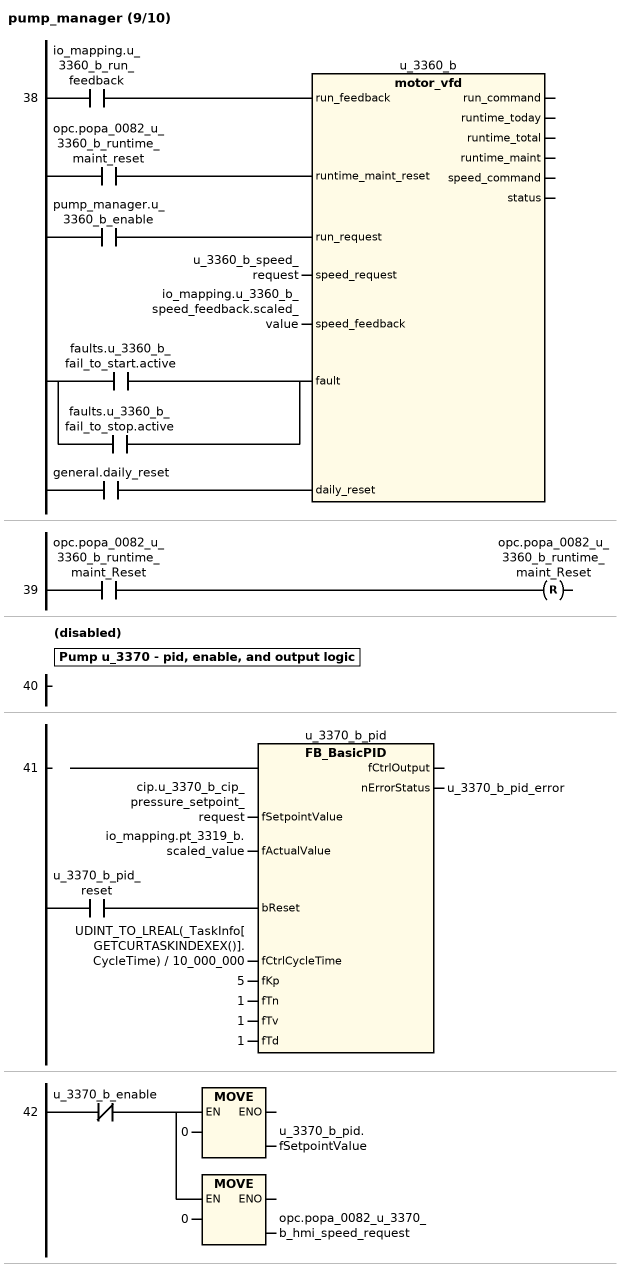
// NETWORK 38
u_3360_b(
    run_feedback := io_mapping.u_3360_b_run_feedback,
    runtime_maint_reset := opc.popa_0082_u_3360_b_runtime_maint_reset,
    run_request := pump_manager.u_3360_b_enable,
    speed_request := u_3360_b_speed_request,
    speed_feedback := io_mapping.u_3360_b_speed_feedback.scaled_value,
    fault := faults.u_3360_b_fail_to_start.active OR faults.u_3360_b_fail_to_stop.active,
    daily_reset := general.daily_reset); // motor_vfd

// NETWORK 39
opc.popa_0082_u_3360_b_runtime_maint_Reset R= opc.popa_0082_u_3360_b_runtime_maint_Reset;

// NETWORK 40 (disabled)
// label: Pump u_3370 - pid, enable, and output logic

// NETWORK 41
u_3370_b_pid(
    fSetpointValue := cip.u_3370_b_cip_pressure_setpoint_request,
    fActualValue := io_mapping.pt_3319_b.scaled_value,
    bReset := u_3370_b_pid_reset,
    fCtrlCycleTime := UDINT_TO_LREAL(_TaskInfo[GETCURTASKINDEXEX()].CycleTime) / 10_000_000,
    fKp := 5,
    fTn := 1,
    fTv := 1,
    fTd := 1,
    nErrorStatus => u_3370_b_pid_error); // FB_BasicPID

// NETWORK 42
_w24 := NOT u_3370_b_enable;
IF _w24 THEN u_3370_b_pid.fSetpointValue := 0; END_IF
IF _w24 THEN opc.popa_0082_u_3370_b_hmi_speed_request := 0; END_IF

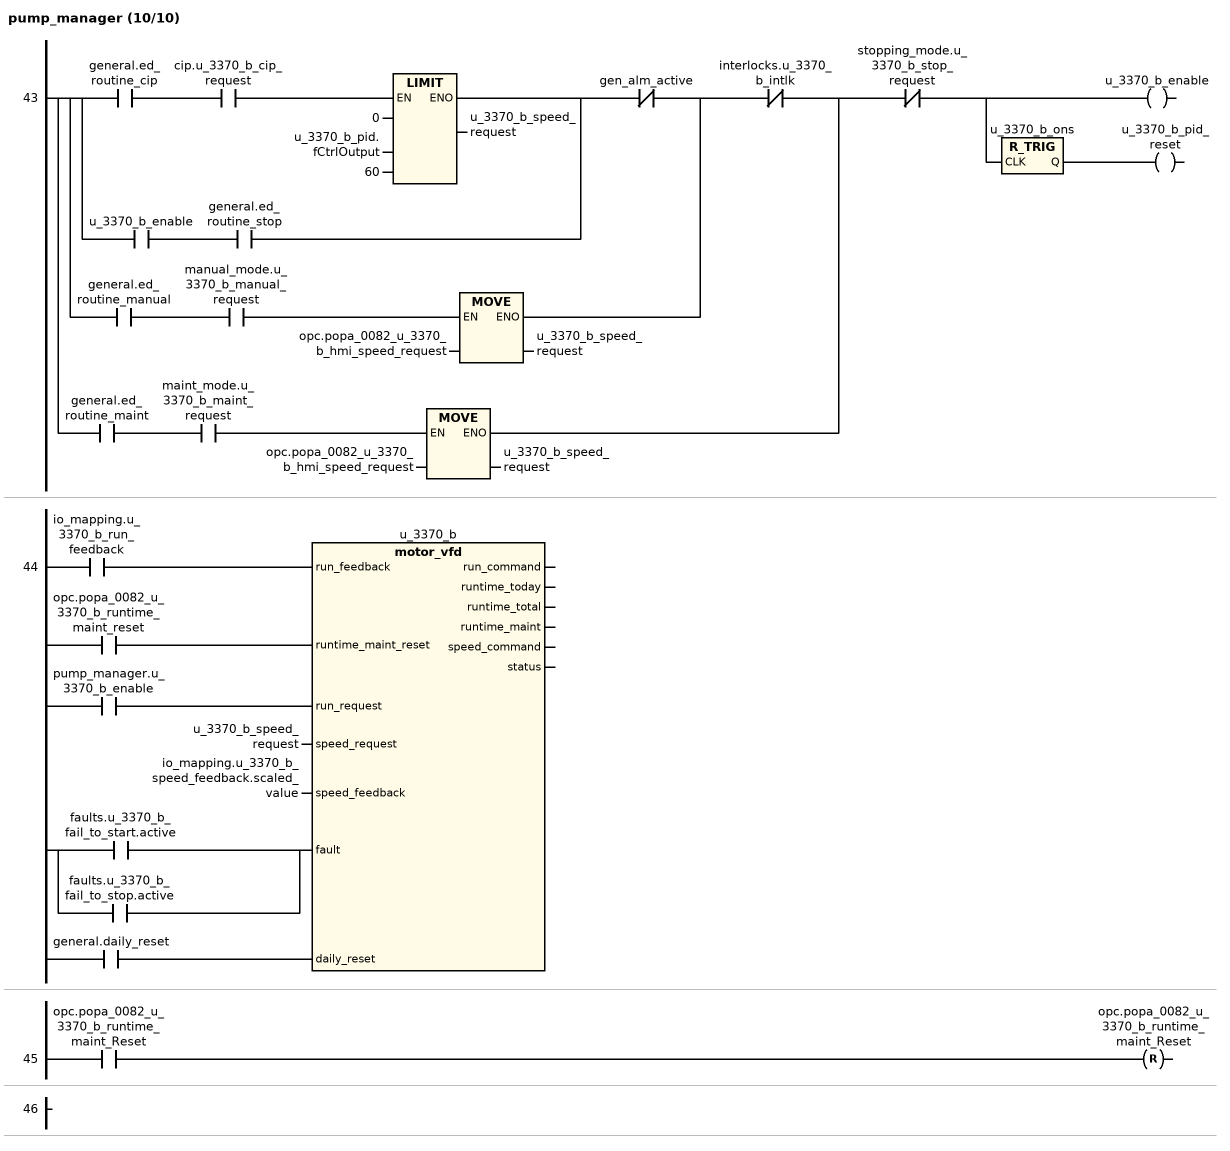
// NETWORK 43
_w25 := general.ed_routine_cip AND cip.u_3370_b_cip_request;
IF _w25 THEN u_3370_b_speed_request := LIMIT(0, u_3370_b_pid.fCtrlOutput, 60); END_IF
_w26 := general.ed_routine_manual AND manual_mode.u_3370_b_manual_request;
IF _w26 THEN u_3370_b_speed_request := opc.popa_0082_u_3370_b_hmi_speed_request; END_IF
_w27 := general.ed_routine_maint AND maint_mode.u_3370_b_maint_request;
IF _w27 THEN u_3370_b_speed_request := opc.popa_0082_u_3370_b_hmi_speed_request; END_IF
_w28 := (((_w25 OR u_3370_b_enable AND general.ed_routine_stop) AND NOT gen_alm_active OR _w26) AND NOT interlocks.u_3370_b_intlk OR _w27) AND NOT stopping_mode.u_3370_b_stop_request;
u_3370_b_enable := _w28;
u_3370_b_ons(CLK := _w28); // R_TRIG
u_3370_b_pid_reset := u_3370_b_ons.Q;

// NETWORK 44
u_3370_b(
    run_feedback := io_mapping.u_3370_b_run_feedback,
    runtime_maint_reset := opc.popa_0082_u_3370_b_runtime_maint_reset,
    run_request := pump_manager.u_3370_b_enable,
    speed_request := u_3370_b_speed_request,
    speed_feedback := io_mapping.u_3370_b_speed_feedback.scaled_value,
    fault := faults.u_3370_b_fail_to_start.active OR faults.u_3370_b_fail_to_stop.active,
    daily_reset := general.daily_reset); // motor_vfd

// NETWORK 45
opc.popa_0082_u_3370_b_runtime_maint_Reset R= opc.popa_0082_u_3370_b_runtime_maint_Reset;

// NETWORK 46

END_PROGRAM

// ---- POUs/idle.TcPOU
PROGRAM idle
VAR
	ed_routine_idle: BOOL;
	redox_doser_idle_enable: BOOL;
	
	tmr_idle_pumps: TON;
	u_3112_a_idle_request: BOOL;
	u_3312_a_idle_request: BOOL;
	u_3405_a_idle_request: BOOL;
	u_3212_a_idle_request: BOOL;
	tmr_idle_pump_delay: TON;
	u_3112_a_running: BOOL;
	u_3112_a_speed_ref: INT;
	u_3112_a_sp: REAL;
	salt_pressure_actual: REAL;
	u_3112_a_ready: BOOL;
	u_3212_a_running: BOOL;
	u_3212_a_ready: BOOL;
	u_3312_a_ready: BOOL;
	u_3312_a_running: BOOL;
	u_3405_a_running: BOOL;
	u_3405_a_ready: BOOL;
	stack_power_enable: BOOL;
	nv_3110_a_open_request: BOOL;
	nv_3210_a_open_request: BOOL;
	nv_3310_a_open_request: BOOL;
	nv_3110_a_open_feedback: BOOL;
	nv_3210_a_open_feedback: BOOL;
	nv_3310_a_open_feedback: BOOL;
	nv_3110_a_idle_request: BOOL;
	nv_3210_a_idle_request: BOOL;
	nv_3310_a_idle_request: BOOL;
	nv_3135_a_idle_request: BOOL;
	nv_3235_a_idle_request: BOOL;
	nv_3335_a_idle_request: BOOL;
	nv_3372_a_idle_request: BOOL;
	nv_3162_a_idle_request: BOOL;

	idle_stack_power_enable: BOOL;
	idle_TEMP_BIT: BOOL;
	tmr_idle_valye_delay: TON;
	tmr_idle_valve_delay: TON;
	tmr_idle_valve_delay_et: TIME;
	tmr_idle_valve_delay_pt: TIME := T#20S;
	tmr_idle_valve_delay_q: BOOL;
	u_3112_a_idle_pressure_setpoint_request: REAL;
	u_3212_a_idle_pressure_setpoint_request: REAL;
	u_3312_a_idle_pressure_setpoint_request: REAL;
	u_3405_a_idle_pressure_setpoint_request: REAL;
	idle_stable: BOOL;
	av_3148_a_idle_position_request: REAL;
	av_3248_a_idle_position_request: REAL;
	av_3348_a_idle_position_request: REAL;
	redox_pressure_calculation: REAL;
	redox_idle_pressure_sp_request: REAL;
	idle_startup_ons: R_TRIG;
END_VAR
VAR // added by the converter: edge detectors and wires of the graphical bodies
    _w1, _w2, _w3, _w4 : BOOL;
END_VAR

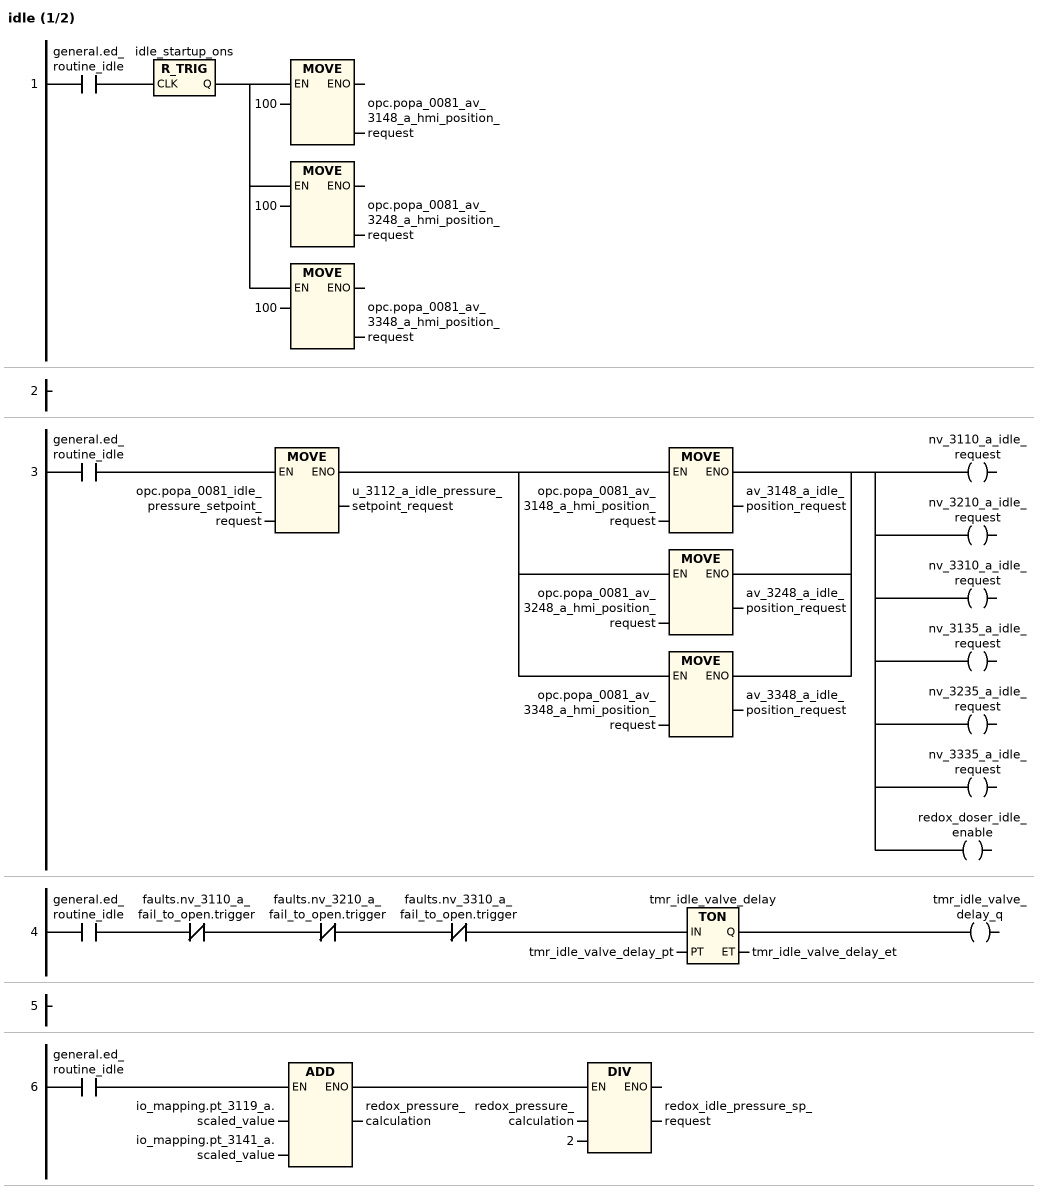
// NETWORK 1
idle_startup_ons(CLK := general.ed_routine_idle); // R_TRIG
IF idle_startup_ons.Q THEN opc.popa_0081_av_3148_a_hmi_position_request := 100; END_IF
IF idle_startup_ons.Q THEN opc.popa_0081_av_3248_a_hmi_position_request := 100; END_IF
IF idle_startup_ons.Q THEN opc.popa_0081_av_3348_a_hmi_position_request := 100; END_IF

// NETWORK 2

// NETWORK 3
_w1 := general.ed_routine_idle;
IF _w1 THEN u_3112_a_idle_pressure_setpoint_request := opc.popa_0081_idle_pressure_setpoint_request; END_IF
IF _w1 THEN av_3148_a_idle_position_request := opc.popa_0081_av_3148_a_hmi_position_request; END_IF
IF _w1 THEN av_3248_a_idle_position_request := opc.popa_0081_av_3248_a_hmi_position_request; END_IF
IF _w1 THEN av_3348_a_idle_position_request := opc.popa_0081_av_3348_a_hmi_position_request; END_IF
_w2 := _w1 OR (_w1 OR _w1);
nv_3110_a_idle_request := _w2;
nv_3210_a_idle_request := _w2;
nv_3310_a_idle_request := _w2;
nv_3135_a_idle_request := _w2;
nv_3235_a_idle_request := _w2;
nv_3335_a_idle_request := _w2;
redox_doser_idle_enable := _w2;

// NETWORK 4
tmr_idle_valve_delay(
    IN := general.ed_routine_idle AND NOT faults.nv_3110_a_fail_to_open.trigger AND NOT faults.nv_3210_a_fail_to_open.trigger AND NOT faults.nv_3310_a_fail_to_open.trigger,
    PT := tmr_idle_valve_delay_pt,
    ET => tmr_idle_valve_delay_et); // TON
tmr_idle_valve_delay_q := tmr_idle_valve_delay.Q;

// NETWORK 5

// NETWORK 6
_w3 := general.ed_routine_idle;
IF _w3 THEN
    redox_pressure_calculation := io_mapping.pt_3119_a.scaled_value + io_mapping.pt_3141_a.scaled_value;
END_IF
IF _w3 THEN redox_idle_pressure_sp_request := redox_pressure_calculation / 2; END_IF

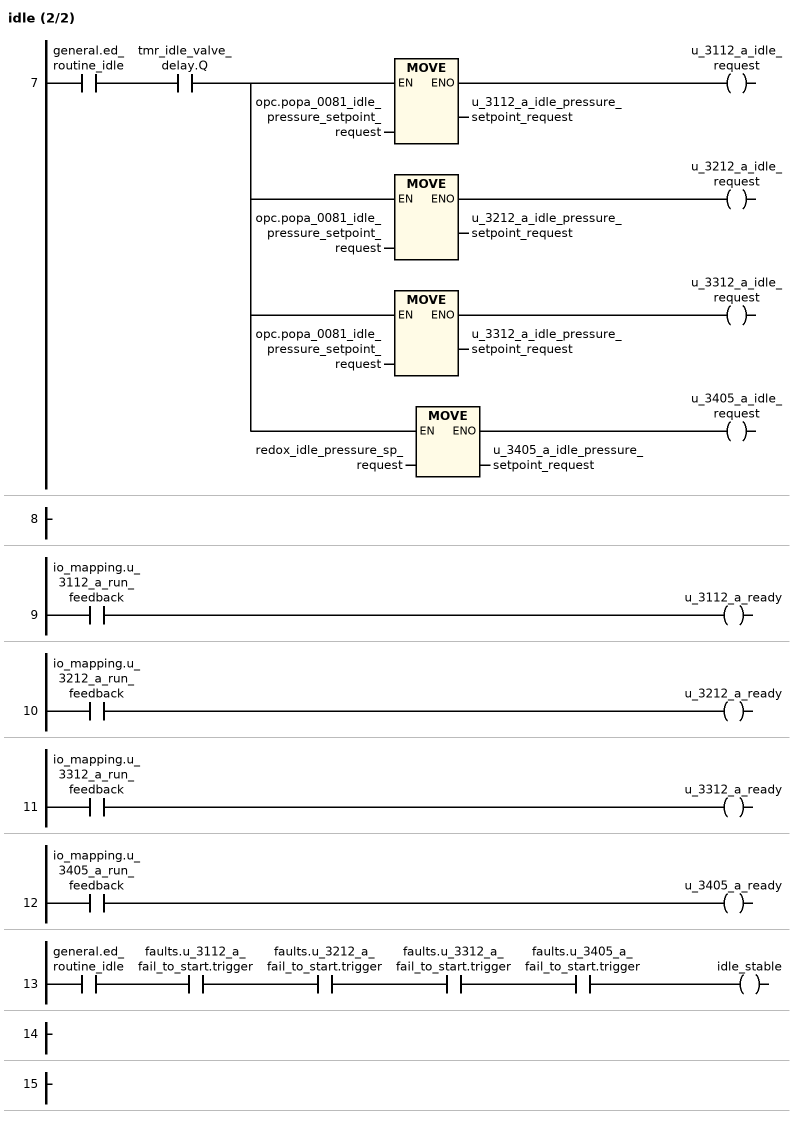
// NETWORK 7
_w4 := general.ed_routine_idle AND tmr_idle_valve_delay.Q;
IF _w4 THEN u_3112_a_idle_pressure_setpoint_request := opc.popa_0081_idle_pressure_setpoint_request; END_IF
u_3112_a_idle_request := _w4;
IF _w4 THEN u_3212_a_idle_pressure_setpoint_request := opc.popa_0081_idle_pressure_setpoint_request; END_IF
u_3212_a_idle_request := _w4;
IF _w4 THEN u_3312_a_idle_pressure_setpoint_request := opc.popa_0081_idle_pressure_setpoint_request; END_IF
u_3312_a_idle_request := _w4;
IF _w4 THEN u_3405_a_idle_pressure_setpoint_request := redox_idle_pressure_sp_request; END_IF
u_3405_a_idle_request := _w4;

// NETWORK 8

// NETWORK 9
u_3112_a_ready := io_mapping.u_3112_a_run_feedback;

// NETWORK 10
u_3212_a_ready := io_mapping.u_3212_a_run_feedback;

// NETWORK 11
u_3312_a_ready := io_mapping.u_3312_a_run_feedback;

// NETWORK 12
u_3405_a_ready := io_mapping.u_3405_a_run_feedback;

// NETWORK 13
idle_stable := general.ed_routine_idle AND faults.u_3112_a_fail_to_start.trigger AND faults.u_3212_a_fail_to_start.trigger AND faults.u_3312_a_fail_to_start.trigger AND faults.u_3405_a_fail_to_start.trigger;

// NETWORK 14

// NETWORK 15

END_PROGRAM

// ---- POUs/general.TcPOU
PROGRAM general
VAR PERSISTENT
	//System date time function block
	system_date_time : date_time;
	//Daily reset bit, used throughout the program for any resets
	daily_reset : BOOL;
	//Alarm Acknoweldge unlatch timer
	alarm_ack_ton : ton;
	//Alarm Reset unlatch timer
	alarm_reset_ton : ton;
	//Alarm Ack and reset unlatch timer setpoint
	alarm_ack_unlatch_sp : TIME :=T#1S;
	
	//Always off bit
	always_off : BOOL := FALSE;
	
	//PLC States - move as needed
	ed_routine_idle : BOOL;
	ed_routine_cip : BOOL;
	ed_routine_manual : BOOL;
	ed_routine_maint : BOOL;
	ed_routine_stop : BOOL;
	ed_critical_stop : BOOL;
	
END_VAR

VAR
	//{attribute 'TcLinkTo' := 'TIID^Device 1 (EtherCAT)^Term 1 (EK1200)^Term 10 (EL2911)^StandardInputs^Standard Out Var 16'}
	twinsafe_safeout AT %I*: BOOL;
	
	//Linked manually
	twinsafe_status AT %I*: USINT;
	twinsafe_reset AT %Q*: BOOL;
	twinsafe_ack AT %Q*: BOOL;
	twinsafe_run AT %Q*: BOOL := TRUE;
	
	test_valve_position AT %I*: INT;
	
	
	test_valve: analog_scaling;
	test_nv_3110_a_open: BOOL;
	safety_reset_ton: TON;
END_VAR
VAR // added by the converter: edge detectors and wires of the graphical bodies
    _rt1, _rt2, _rt3, _rt4, _rt5 : R_TRIG;
    _w1, _w2, _w3, _w4 : BOOL;
END_VAR

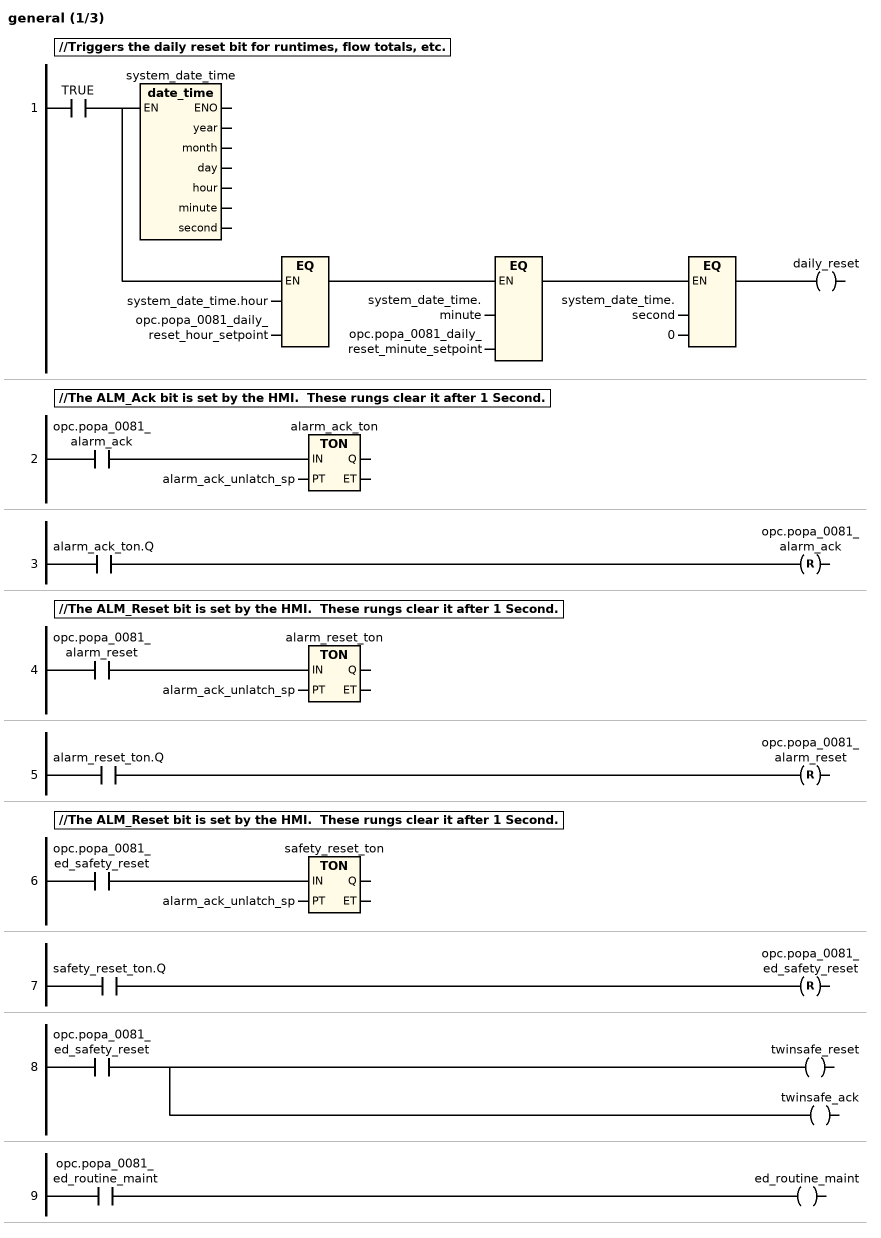
// NETWORK 1
// label: //Triggers the daily reset bit for runtimes, flow totals, etc.
system_date_time(); // date_time
daily_reset := system_date_time.hour = opc.popa_0081_daily_reset_hour_setpoint AND system_date_time.minute = opc.popa_0081_daily_reset_minute_setpoint AND system_date_time.second = 0;

// NETWORK 2
// label: //The ALM_Ack bit is set by the HMI.  These rungs clear it after 1 Second.
alarm_ack_ton(IN := opc.popa_0081_alarm_ack, PT := alarm_ack_unlatch_sp); // TON

// NETWORK 3
opc.popa_0081_alarm_ack R= alarm_ack_ton.Q;

// NETWORK 4
// label: //The ALM_Reset bit is set by the HMI.  These rungs clear it after 1 Second.
alarm_reset_ton(IN := opc.popa_0081_alarm_reset, PT := alarm_ack_unlatch_sp); // TON

// NETWORK 5
opc.popa_0081_alarm_reset R= alarm_reset_ton.Q;

// NETWORK 6
// label: //The ALM_Reset bit is set by the HMI.  These rungs clear it after 1 Second.
safety_reset_ton(IN := opc.popa_0081_ed_safety_reset, PT := alarm_ack_unlatch_sp); // TON

// NETWORK 7
opc.popa_0081_ed_safety_reset R= safety_reset_ton.Q;

// NETWORK 8
twinsafe_reset := opc.popa_0081_ed_safety_reset;
twinsafe_ack := opc.popa_0081_ed_safety_reset;

// NETWORK 9
ed_routine_maint := opc.popa_0081_ed_routine_maint;

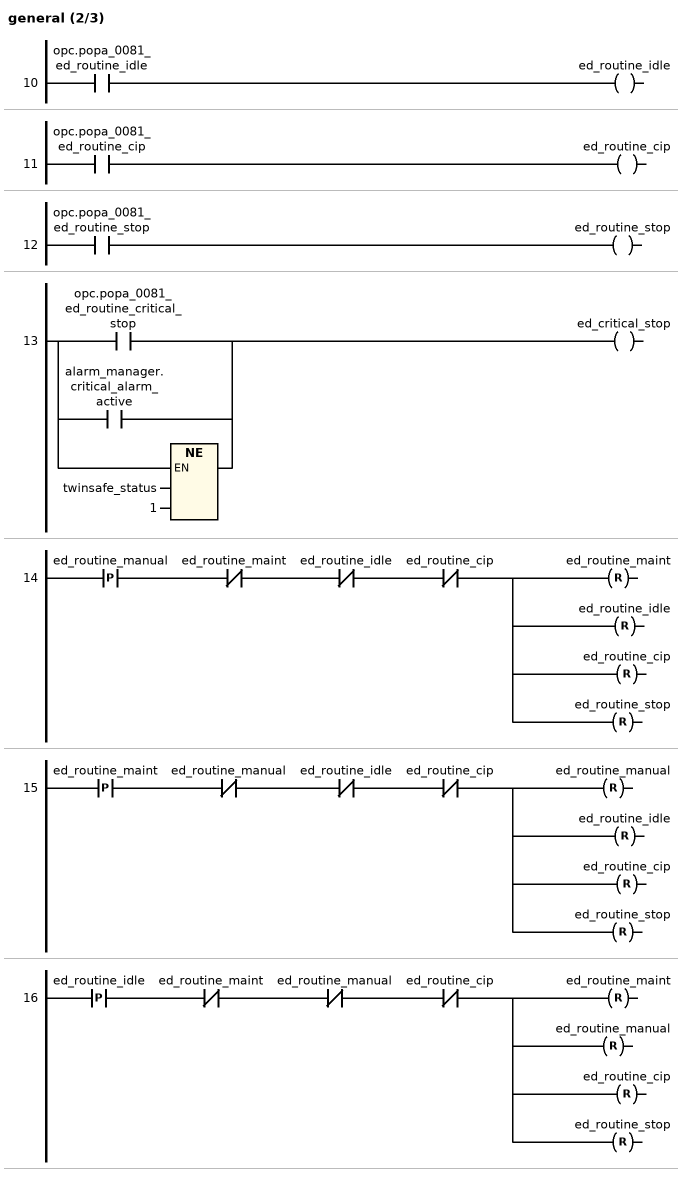
// NETWORK 10
ed_routine_idle := opc.popa_0081_ed_routine_idle;

// NETWORK 11
ed_routine_cip := opc.popa_0081_ed_routine_cip;

// NETWORK 12
ed_routine_stop := opc.popa_0081_ed_routine_stop;

// NETWORK 13
ed_critical_stop := opc.popa_0081_ed_routine_critical_stop OR alarm_manager.critical_alarm_active OR twinsafe_status <> 1;

// NETWORK 14
_rt1(CLK := ed_routine_manual);
_w1 := _rt1.Q AND NOT ed_routine_maint AND NOT ed_routine_idle AND NOT ed_routine_cip;
ed_routine_maint R= _w1;
ed_routine_idle R= _w1;
ed_routine_cip R= _w1;
ed_routine_stop R= _w1;

// NETWORK 15
_rt2(CLK := ed_routine_maint);
_w2 := _rt2.Q AND NOT ed_routine_manual AND NOT ed_routine_idle AND NOT ed_routine_cip;
ed_routine_manual R= _w2;
ed_routine_idle R= _w2;
ed_routine_cip R= _w2;
ed_routine_stop R= _w2;

// NETWORK 16
_rt3(CLK := ed_routine_idle);
_w3 := _rt3.Q AND NOT ed_routine_maint AND NOT ed_routine_manual AND NOT ed_routine_cip;
ed_routine_maint R= _w3;
ed_routine_manual R= _w3;
ed_routine_cip R= _w3;
ed_routine_stop R= _w3;

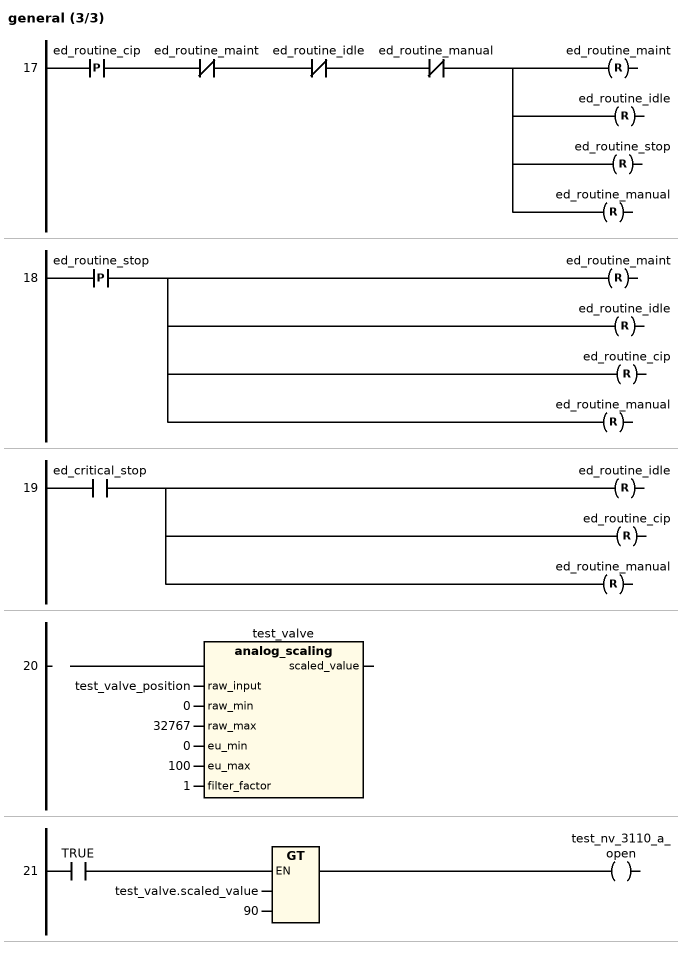
// NETWORK 17
_rt4(CLK := ed_routine_cip);
_w4 := _rt4.Q AND NOT ed_routine_maint AND NOT ed_routine_idle AND NOT ed_routine_manual;
ed_routine_maint R= _w4;
ed_routine_idle R= _w4;
ed_routine_stop R= _w4;
ed_routine_manual R= _w4;

// NETWORK 18
_rt5(CLK := ed_routine_stop);
ed_routine_maint R= _rt5.Q;
ed_routine_idle R= _rt5.Q;
ed_routine_cip R= _rt5.Q;
ed_routine_manual R= _rt5.Q;

// NETWORK 19
ed_routine_idle R= ed_critical_stop;
ed_routine_cip R= ed_critical_stop;
ed_routine_manual R= ed_critical_stop;

// NETWORK 20
test_valve(
    raw_input := test_valve_position,
    raw_min := 0,
    raw_max := 32767,
    eu_min := 0,
    eu_max := 100,
    filter_factor := 1); // analog_scaling

// NETWORK 21
test_nv_3110_a_open := test_valve.scaled_value > 90;

END_PROGRAM

// ---- POUs/Function Blocks/analog_scaling.TcPOU
FUNCTION_BLOCK analog_scaling
VAR_INPUT
	//Raw Input value
	raw_input : REAL;
	//Raw Input Minimum Scaling Value
	raw_min : REAL :=0;
	//Raw Input Maximum Scaling Value
	raw_max : REAL :=32767;
	//Engineering Units Minimum Scaling Value
	eu_min : REAL;
	//Engineering Units Maximum Scaling Value
	eu_max : REAL;
	//Averaging Filter Time Setpoint
	filter_factor : REAL;
END_VAR
VAR_OUTPUT
	//Scaled Value for Output
	scaled_value : REAL;
END_VAR
VAR
	//Scratchpad Value
	normalized_value : REAL;
	//unfiltered Scaled Value
	unfiltered_value : REAL;
END_VAR

//Initialize Raw_Max and EU_Max to avoid Scaled_Value=Not a number
IF raw_max = 0 AND raw_min = 0 THEN
	raw_max:=1;
END_IF
IF eu_max = 0 AND eu_min = 0 THEN
	eu_max:=1;
END_IF

//Normalize the Analog Input
IF raw_input < raw_min THEN
		normalized_value := raw_min;
	ELSIF raw_input > raw_max THEN
		normalized_value := raw_max;
	ELSE
		normalized_value := (raw_input - raw_min) / (raw_max - raw_min);
	END_IF
	
//Scale the Output
unfiltered_value := normalized_value * (eu_max-eu_min)+eu_min;

//Low Pass Filter for the output.  Increase Filter to dampen reading
scaled_value := ((scaled_value * filter_factor) + unfiltered_value) / (filter_factor +1);

END_FUNCTION_BLOCK

// ---- POUs/io_mapping.TcPOU
PROGRAM io_mapping
VAR PERSISTENT
//---Field Instrumentation-----------------------------------------------------------------------------------------------
    //Analog input function block
	cpt_3144_b: analog_scaling;
	
	cct_3120_b : analog_scaling;
	cct_3220_b : analog_scaling;
	cct_3320_b : analog_scaling;
	cct_3142_b : analog_scaling;
	cct_3242_b : analog_scaling;
	cct_3342_b : analog_scaling;
	
	ft_3122_b : analog_scaling;
	ft_3222_b : analog_scaling;
	ft_3322_b : analog_scaling;
	
	lt_3102_b : analog_scaling;
	lt_3202_b : analog_scaling;
	lt_3302_b : analog_scaling;
	lt_3153_b : analog_scaling;
	lt_3253_b : analog_scaling;
	lt_3353_b : analog_scaling;
	lt_3402_b : analog_scaling;
	
    pt_3119_b : analog_scaling;
	pt_3219_b : analog_scaling;
	pt_3319_b : analog_scaling;
	pt_3141_b : analog_scaling;
	pt_3241_b : analog_scaling;
	pt_3341_b : analog_scaling;
	pt_3428_b : analog_scaling;
	pt_3414_b : analog_scaling;
	
	tt_3118_b : analog_scaling;
	tt_3218_b : analog_scaling;
	tt_3318_b : analog_scaling;
	tt_3140_b : analog_scaling;
	tt_3240_b : analog_scaling;
	tt_3340_b : analog_scaling;
	tt_3432_b : analog_scaling;

	//Motor vfd speed feedback
	u_3112_b_speed_feedback : analog_scaling;
	u_3212_b_speed_feedback : analog_scaling;
	u_3312_b_speed_feedback : analog_scaling;
	u_3160_b_speed_feedback : analog_scaling;
	u_3260_b_speed_feedback : analog_scaling;
	u_3360_b_speed_feedback : analog_scaling;
	u_3370_b_speed_feedback : analog_scaling;
	u_3405_b_speed_feedback : analog_scaling;	
	
	//Analog valve position feedback
	av_3148_b_position_feedback : analog_scaling;
	av_3248_b_position_feedback : analog_scaling;
	av_3348_b_position_feedback : analog_scaling;
    //Analog input raw input, mapped to a physical input
    cpt_3144_b_raw_input AT %I* : INT;
	{attribute 'TcLinkTo' := 'TIID^Device 1 (EtherCAT)^Term 20 (EK1100-0018)^Term 24 (EL3058)^AI Standard Channel 1^Value'}
	cct_3120_b_raw_input AT %I* : INT;
	{attribute 'TcLinkTo' := 'TIID^Device 1 (EtherCAT)^Term 20 (EK1100-0018)^Term 24 (EL3058)^AI Standard Channel 2^Value'}
	cct_3220_b_raw_input AT %I* : INT;
	{attribute 'TcLinkTo' := 'TIID^Device 1 (EtherCAT)^Term 20 (EK1100-0018)^Term 24 (EL3058)^AI Standard Channel 3^Value'}
	cct_3320_b_raw_input AT %I* : INT;
	{attribute 'TcLinkTo' := 'TIID^Device 1 (EtherCAT)^Term 20 (EK1100-0018)^Term 24 (EL3058)^AI Standard Channel 4^Value'}
	cct_3142_b_raw_input AT %I* : INT;
	{attribute 'TcLinkTo' := 'TIID^Device 1 (EtherCAT)^Term 20 (EK1100-0018)^Term 24 (EL3058)^AI Standard Channel 5^Value'}
	cct_3242_b_raw_input AT %I* : INT;
	{attribute 'TcLinkTo' := 'TIID^Device 1 (EtherCAT)^Term 20 (EK1100-0018)^Term 24 (EL3058)^AI Standard Channel 6^Value'}
	cct_3342_b_raw_input AT %I* : INT;
	
	{attribute 'TcLinkTo' := 'TIID^Device 1 (EtherCAT)^Term 20 (EK1100-0018)^Term 25 (EL3058)^AI Standard Channel 1^Value'}
	ft_3122_b_raw_input AT %I* : INT;
	{attribute 'TcLinkTo' := 'TIID^Device 1 (EtherCAT)^Term 20 (EK1100-0018)^Term 25 (EL3058)^AI Standard Channel 2^Value'}
	ft_3222_b_raw_input AT %I* : INT;
	{attribute 'TcLinkTo' := 'TIID^Device 1 (EtherCAT)^Term 20 (EK1100-0018)^Term 25 (EL3058)^AI Standard Channel 3^Value'}
	ft_3322_b_raw_input AT %I* : INT;
	
	{attribute 'TcLinkTo' := 'TIID^Device 1 (EtherCAT)^Term 20 (EK1100-0018)^Term 21 (EL3058)^AI Standard Channel 1^Value'}
	pt_3119_b_raw_input AT %I* : INT;
	{attribute 'TcLinkTo' := 'TIID^Device 1 (EtherCAT)^Term 20 (EK1100-0018)^Term 21 (EL3058)^AI Standard Channel 2^Value'}
	pt_3219_b_raw_input AT %I* : INT;
	{attribute 'TcLinkTo' := 'TIID^Device 1 (EtherCAT)^Term 20 (EK1100-0018)^Term 21 (EL3058)^AI Standard Channel 3^Value'}
	pt_3319_b_raw_input AT %I* : INT;
	{attribute 'TcLinkTo' := 'TIID^Device 1 (EtherCAT)^Term 20 (EK1100-0018)^Term 21 (EL3058)^AI Standard Channel 4^Value'}
	pt_3141_b_raw_input AT %I* : INT;
	{attribute 'TcLinkTo' := 'TIID^Device 1 (EtherCAT)^Term 20 (EK1100-0018)^Term 21 (EL3058)^AI Standard Channel 5^Value'}
	pt_3241_b_raw_input AT %I* : INT;
	{attribute 'TcLinkTo' := 'TIID^Device 1 (EtherCAT)^Term 20 (EK1100-0018)^Term 21 (EL3058)^AI Standard Channel 6^Value'}
	pt_3341_b_raw_input AT %I* : INT;
	{attribute 'TcLinkTo' := 'TIID^Device 1 (EtherCAT)^Term 40 (EK1100)^Term 41 (EL3058)^AI Standard Channel 4^Value'}
	pt_3428_b_raw_input AT %I* : INT;
	{attribute 'TcLinkTo' := 'TIID^Device 1 (EtherCAT)^Term 40 (EK1100)^Term 41 (EL3058)^AI Standard Channel 5^Value'}
	pt_3414_b_raw_input AT %I* : INT;
	
	{attribute 'TcLinkTo' := 'TIID^Device 1 (EtherCAT)^Term 20 (EK1100-0018)^Term 23 (EL3058)^AI Standard Channel 3^Value'}
	lt_3102_b_raw_input AT %I* : INT;
	{attribute 'TcLinkTo' := 'TIID^Device 1 (EtherCAT)^Term 20 (EK1100-0018)^Term 23 (EL3058)^AI Standard Channel 4^Value'}
	lt_3202_b_raw_input AT %I* : INT;
	{attribute 'TcLinkTo' := 'TIID^Device 1 (EtherCAT)^Term 20 (EK1100-0018)^Term 23 (EL3058)^AI Standard Channel 5^Value'}
	lt_3302_b_raw_input AT %I* : INT;
	{attribute 'TcLinkTo' := 'TIID^Device 1 (EtherCAT)^Term 20 (EK1100-0018)^Term 23 (EL3058)^AI Standard Channel 6^Value'}
	lt_3153_b_raw_input AT %I* : INT;
	{attribute 'TcLinkTo' := 'TIID^Device 1 (EtherCAT)^Term 20 (EK1100-0018)^Term 23 (EL3058)^AI Standard Channel 7^Value'}
	lt_3253_b_raw_input AT %I* : INT;
	{attribute 'TcLinkTo' := 'TIID^Device 1 (EtherCAT)^Term 20 (EK1100-0018)^Term 23 (EL3058)^AI Standard Channel 8^Value'}
	lt_3353_b_raw_input AT %I* : INT;
	{attribute 'TcLinkTo' := 'TIID^Device 1 (EtherCAT)^Term 40 (EK1100)^Term 41 (EL3058)^AI Standard Channel 3^Value'}
	lt_3402_b_raw_input AT %I* : INT;
	
	{attribute 'TcLinkTo' := 'TIID^Device 1 (EtherCAT)^Term 20 (EK1100-0018)^Term 21 (EL3058)^AI Standard Channel 7^Value'}
	tt_3118_b_raw_input AT %I* : INT;
	{attribute 'TcLinkTo' := 'TIID^Device 1 (EtherCAT)^Term 20 (EK1100-0018)^Term 21 (EL3058)^AI Standard Channel 8^Value'}
	tt_3218_b_raw_input AT %I* : INT;
	{attribute 'TcLinkTo' := 'TIID^Device 1 (EtherCAT)^Term 20 (EK1100-0018)^Term 22 (EL3058)^AI Standard Channel 1^Value'}
	tt_3318_b_raw_input AT %I* : INT;
	{attribute 'TcLinkTo' := 'TIID^Device 1 (EtherCAT)^Term 20 (EK1100-0018)^Term 22 (EL3058)^AI Standard Channel 2^Value'}
	tt_3140_b_raw_input AT %I* : INT;
	{attribute 'TcLinkTo' := 'TIID^Device 1 (EtherCAT)^Term 20 (EK1100-0018)^Term 22 (EL3058)^AI Standard Channel 3^Value'}
	tt_3240_b_raw_input AT %I* : INT;
	{attribute 'TcLinkTo' := 'TIID^Device 1 (EtherCAT)^Term 20 (EK1100-0018)^Term 22 (EL3058)^AI Standard Channel 4^Value'}
	tt_3340_b_raw_input AT %I* : INT;
	{attribute 'TcLinkTo' := 'TIID^Device 1 (EtherCAT)^Term 40 (EK1100)^Term 41 (EL3058)^AI Standard Channel 2^Value'}
	tt_3432_b_raw_input AT %I* : INT;
	
//---Field Equipment:Pumps----------------------------------------------------------------------------------------------------------
	
	//Motor vfd run feedback, mapped to a physical input
	{attribute 'TcLinkTo' := 'TIID^Device 1 (EtherCAT)^Term 1 (EK1200)^Term 7 (EL1859)^Channel 2^Input'}
	u_3112_b_run_feedback AT %I* : BOOL;
	{attribute 'TcLinkTo' := 'TIID^Device 1 (EtherCAT)^Term 1 (EK1200)^Term 7 (EL1859)^Channel 4^Input'}
	u_3212_b_run_feedback AT %I* : BOOL;
	{attribute 'TcLinkTo' := 'TIID^Device 1 (EtherCAT)^Term 1 (EK1200)^Term 7 (EL1859)^Channel 6^Input'}
	u_3312_b_run_feedback AT %I* : BOOL;
	{attribute 'TcLinkTo' := 'TIID^Device 1 (EtherCAT)^Term 1 (EK1200)^Term 7 (EL1859)^Channel 8^Input'}
	u_3160_b_run_feedback AT %I* : BOOL;
	{attribute 'TcLinkTo' := 'TIID^Device 1 (EtherCAT)^Term 1 (EK1200)^Term 8 (EL1859)^Channel 2^Input'}
	u_3260_b_run_feedback AT %I* : BOOL;
	{attribute 'TcLinkTo' := 'TIID^Device 1 (EtherCAT)^Term 1 (EK1200)^Term 8 (EL1859)^Channel 4^Input'}
	u_3360_b_run_feedback AT %I* : BOOL;
	{attribute 'TcLinkTo' := 'TIID^Device 1 (EtherCAT)^Term 1 (EK1200)^Term 8 (EL1859)^Channel 6^Input'}
	u_3370_b_run_feedback AT %I* : BOOL;
	{attribute 'TcLinkTo' := 'TIID^Device 1 (EtherCAT)^Term 40 (EK1100)^Term 43 (EL1859)^Channel 2^Input'}
	u_3405_b_run_feedback AT %I* : BOOL;
	
	//Motor Fault feedback
	{attribute 'TcLinkTo' := 'TIID^Device 1 (EtherCAT)^Term 1 (EK1200)^Term 7 (EL1859)^Channel 1^Input'}
	u_3112_b_fault_feedback AT %I* : BOOL;
	{attribute 'TcLinkTo' := 'TIID^Device 1 (EtherCAT)^Term 1 (EK1200)^Term 7 (EL1859)^Channel 3^Input'}
	u_3212_b_fault_feedback AT %I* : BOOL;
	{attribute 'TcLinkTo' := 'TIID^Device 1 (EtherCAT)^Term 1 (EK1200)^Term 7 (EL1859)^Channel 5^Input'}
	u_3312_b_fault_feedback AT %I* : BOOL;
	{attribute 'TcLinkTo' := 'TIID^Device 1 (EtherCAT)^Term 1 (EK1200)^Term 7 (EL1859)^Channel 7^Input'}
	u_3160_b_fault_feedback AT %I* : BOOL;
	{attribute 'TcLinkTo' := 'TIID^Device 1 (EtherCAT)^Term 1 (EK1200)^Term 8 (EL1859)^Channel 1^Input'}
	u_3260_b_fault_feedback AT %I* : BOOL;
	{attribute 'TcLinkTo' := 'TIID^Device 1 (EtherCAT)^Term 1 (EK1200)^Term 8 (EL1859)^Channel 3^Input'}
	u_3360_b_fault_feedback AT %I* : BOOL;
	{attribute 'TcLinkTo' := 'TIID^Device 1 (EtherCAT)^Term 1 (EK1200)^Term 8 (EL1859)^Channel 5^Input'}
	u_3370_b_fault_feedback AT %I* : BOOL;
	{attribute 'TcLinkTo' := 'TIID^Device 1 (EtherCAT)^Term 40 (EK1100)^Term 43 (EL1859)^Channel 1^Input'}
	u_3405_b_fault_feedback AT %I* : BOOL;
	
	
	
	

	
	//Motor vfd speed feedback raw input
	{attribute 'TcLinkTo' := 'TIID^Device 1 (EtherCAT)^Term 1 (EK1200)^Term 2 (EL3058)^AI Standard Channel 1^Value'}
	u_3112_b_speed_feedback_raw_input AT %I* : INT;
	{attribute 'TcLinkTo' := 'TIID^Device 1 (EtherCAT)^Term 1 (EK1200)^Term 2 (EL3058)^AI Standard Channel 2^Value'}
	u_3212_b_speed_feedback_raw_input AT %I* : INT;
	{attribute 'TcLinkTo' := 'TIID^Device 1 (EtherCAT)^Term 1 (EK1200)^Term 2 (EL3058)^AI Standard Channel 3^Value'}
	u_3312_b_speed_feedback_raw_input AT %I* : INT;
	{attribute 'TcLinkTo' := 'TIID^Device 1 (EtherCAT)^Term 1 (EK1200)^Term 2 (EL3058)^AI Standard Channel 4^Value'}
	u_3160_b_speed_feedback_raw_input AT %I* : INT;
	{attribute 'TcLinkTo' := 'TIID^Device 1 (EtherCAT)^Term 1 (EK1200)^Term 2 (EL3058)^AI Standard Channel 5^Value'}
	u_3260_b_speed_feedback_raw_input AT %I* : INT;
	{attribute 'TcLinkTo' := 'TIID^Device 1 (EtherCAT)^Term 1 (EK1200)^Term 2 (EL3058)^AI Standard Channel 6^Value'}
	u_3360_b_speed_feedback_raw_input AT %I* : INT;
	{attribute 'TcLinkTo' := 'TIID^Device 1 (EtherCAT)^Term 1 (EK1200)^Term 2 (EL3058)^AI Standard Channel 7^Value'}
	u_3370_b_speed_feedback_raw_input AT %I* : INT;
	{attribute 'TcLinkTo' := 'TIID^Device 1 (EtherCAT)^Term 40 (EK1100)^Term 41 (EL3058)^AI Standard Channel 1^Value'}
	u_3405_b_speed_feedback_raw_input AT %I* : INT;
	
//--Field Equipent: Valves---------------------------------------------------------------------------------------------------------------
	

	//Analog valve position feedback raw input
	{attribute 'TcLinkTo' := 'TIID^Device 1 (EtherCAT)^Term 20 (EK1100-0018)^Term 22 (EL3058)^AI Standard Channel 8^Value'}
	av_3148_b_position_feedback_raw_input AT %I* : INT;
	{attribute 'TcLinkTo' := 'TIID^Device 1 (EtherCAT)^Term 20 (EK1100-0018)^Term 23 (EL3058)^AI Standard Channel 1^Value'}
	av_3248_b_position_feedback_raw_input AT %I* : INT;
	{attribute 'TcLinkTo' := 'TIID^Device 1 (EtherCAT)^Term 20 (EK1100-0018)^Term 23 (EL3058)^AI Standard Channel 2^Value'}
	av_3348_b_position_feedback_raw_input AT %I* : INT;
	

	
	//Digital valve open feedback
	//{attribute 'TcLinkTo' := 'TIID^Device 1 (EtherCAT)^Term 31 (EK1914)^Term 32 (EL1859)^Channel 11^Output'}
	nv_3110_b_open_feedback AT %I* : BOOL;
	//{attribute 'TcLinkTo' := 'TIID^Device 1 (EtherCAT)^Term 31 (EK1914)^Term 32 (EL1859)^Channel 11^Output'}
	nv_3210_b_open_feedback AT %I* : BOOL;
	//{attribute 'TcLinkTo' := 'TIID^Device 1 (EtherCAT)^Term 31 (EK1914)^Term 32 (EL1859)^Channel 11^Output'}
	nv_3310_b_open_feedback AT %I* : BOOL;
	{attribute 'TcLinkTo' := 'TIID^Device 1 (EtherCAT)^Term 20 (EK1100-0018)^Term 28 (EL1859)^Channel 1^Input'}
	nv_3135_b_open_feedback AT %I* : BOOL;
	{attribute 'TcLinkTo' := 'TIID^Device 1 (EtherCAT)^Term 20 (EK1100-0018)^Term 28 (EL1859)^Channel 2^Input'}
	nv_3235_b_open_feedback AT %I* : BOOL;
	{attribute 'TcLinkTo' := 'TIID^Device 1 (EtherCAT)^Term 20 (EK1100-0018)^Term 28 (EL1859)^Channel 3^Input'}
	nv_3335_b_open_feedback AT %I* : BOOL;
	{attribute 'TcLinkTo' := 'TIID^Device 1 (EtherCAT)^Term 20 (EK1100-0018)^Term 28 (EL1859)^Channel 4^Input'}
	nv_3372_b_open_feedback AT %I* : BOOL;
	{attribute 'TcLinkTo' := 'TIID^Device 1 (EtherCAT)^Term 20 (EK1100-0018)^Term 28 (EL1859)^Channel 5^Input'}
	nv_3162_b_open_feedback AT %I* : BOOL;
	
	//Digital valve closed feedback
	//{attribute 'TcLinkTo' := 'TIID^Device 1 (EtherCAT)^Term 31 (EK1914)^Term 32 (EL1859)^Channel 11^Output'}
	nv_3110_b_closed_feedback AT %I* : BOOL;
	//{attribute 'TcLinkTo' := 'TIID^Device 1 (EtherCAT)^Term 31 (EK1914)^Term 32 (EL1859)^Channel 11^Output'}
	nv_3210_b_closed_feedback AT %I* : BOOL;
	//{attribute 'TcLinkTo' := 'TIID^Device 1 (EtherCAT)^Term 31 (EK1914)^Term 32 (EL1859)^Channel 11^Output'}
	nv_3310_b_closed_feedback AT %I* : BOOL;
	{attribute 'TcLinkTo' := 'TIID^Device 1 (EtherCAT)^Term 20 (EK1100-0018)^Term 29 (EL1859)^Channel 1^Input'}
	nv_3135_b_closed_feedback AT %I* : BOOL;
	{attribute 'TcLinkTo' := 'TIID^Device 1 (EtherCAT)^Term 20 (EK1100-0018)^Term 29 (EL1859)^Channel 2^Input'}
	nv_3235_b_closed_feedback AT %I* : BOOL;
	{attribute 'TcLinkTo' := 'TIID^Device 1 (EtherCAT)^Term 20 (EK1100-0018)^Term 29 (EL1859)^Channel 3^Input'}
	nv_3335_b_closed_feedback AT %I* : BOOL;
	{attribute 'TcLinkTo' := 'TIID^Device 1 (EtherCAT)^Term 20 (EK1100-0018)^Term 29 (EL1859)^Channel 4^Input'}
	nv_3372_b_closed_feedback AT %I* : BOOL;
	{attribute 'TcLinkTo' := 'TIID^Device 1 (EtherCAT)^Term 20 (EK1100-0018)^Term 29 (EL1859)^Channel 5^Input'}
	nv_3162_b_closed_feedback AT %I* : BOOL;
	

END_VAR

//---Field Instrumentation--------------------------------------------------------------------------------------------------

//Instantiate analog input function block
cpt_3144_b();
//Map values from the OPC GVL so that they can be written to from outside POU(IE from HMI)
cpt_3144_b.eu_max:=opc.popa_0082_cpt_3144_b_eu_max;
cpt_3144_b.eu_min:=opc.popa_0082_cpt_3144_b_eu_min;
cpt_3144_b.filter_factor:=opc.popa_0082_cpt_3144_b_filter_factor;
cpt_3144_b.raw_max:=opc.popa_0082_cpt_3144_b_raw_max;
cpt_3144_b.raw_min:=opc.popa_0082_cpt_3144_b_raw_min;
//Map the analog scaling function block raw input to the physical raw input variable
cpt_3144_b.raw_input := cpt_3144_b_raw_input;

//Instantiate analog input function block
cct_3120_b();
//Map values from the OPC GVL so that they can be written to from outside POU(IE from HMI)
cct_3120_b.eu_max:=opc.popa_0082_cct_3120_b_eu_max;
cct_3120_b.eu_min:=opc.popa_0082_cct_3120_b_eu_min;
cct_3120_b.filter_factor:=opc.popa_0082_cct_3120_b_filter_factor;
cct_3120_b.raw_max:=opc.popa_0082_cct_3120_b_raw_max;
cct_3120_b.raw_min:=opc.popa_0082_cct_3120_b_raw_min;
//Map the analog scaling function block raw input to the physical raw input variable
cct_3120_b.raw_input := cct_3120_b_raw_input;

//Instantiate analog input function block
cct_3220_b();
//Map values from the OPC GVL so that they can be written to from outside POU(IE from HMI)
cct_3220_b.eu_max:=opc.popa_0082_cct_3220_b_eu_max;
cct_3220_b.eu_min:=opc.popa_0082_cct_3220_b_eu_min;
cct_3220_b.filter_factor:=opc.popa_0082_cct_3220_b_filter_factor;
cct_3220_b.raw_max:=opc.popa_0082_cct_3220_b_raw_max;
cct_3220_b.raw_min:=opc.popa_0082_cct_3220_b_raw_min;
//Map the analog scaling function block raw input to the physical raw input variable
cct_3220_b.raw_input := cct_3220_b_raw_input;

//Instantiate analog input function block
cct_3320_b();
//Map values from the OPC GVL so that they can be written to from outside POU(IE from HMI)
cct_3320_b.eu_max:=opc.popa_0082_cct_3320_b_eu_max;
cct_3320_b.eu_min:=opc.popa_0082_cct_3320_b_eu_min;
cct_3320_b.filter_factor:=opc.popa_0082_cct_3320_b_filter_factor;
cct_3320_b.raw_max:=opc.popa_0082_cct_3320_b_raw_max;
cct_3320_b.raw_min:=opc.popa_0082_cct_3320_b_raw_min;
//Map the analog scaling function block raw input to the physical raw input variable
cct_3320_b.raw_input := cct_3320_b_raw_input;

//Instantiate analog input function block
cct_3142_b();
//Map values from the OPC GVL so that they can be written to from outside POU(IE from HMI)
cct_3142_b.eu_max:=opc.popa_0082_cct_3142_b_eu_max;
cct_3142_b.eu_min:=opc.popa_0082_cct_3142_b_eu_min;
cct_3142_b.filter_factor:=opc.popa_0082_cct_3142_b_filter_factor;
cct_3142_b.raw_max:=opc.popa_0082_cct_3142_b_raw_max;
cct_3142_b.raw_min:=opc.popa_0082_cct_3142_b_raw_min;
//Map the analog scaling function block raw input to the physical raw input variable
cct_3142_b.raw_input := cct_3142_b_raw_input;

//Instantiate analog input function block
cct_3242_b();
//Map values from the OPC GVL so that they can be written to from outside POU(IE from HMI)
cct_3242_b.eu_max:=opc.popa_0082_cct_3242_b_eu_max;
cct_3242_b.eu_min:=opc.popa_0082_cct_3242_b_eu_min;
cct_3242_b.filter_factor:=opc.popa_0082_cct_3242_b_filter_factor;
cct_3242_b.raw_max:=opc.popa_0082_cct_3242_b_raw_max;
cct_3242_b.raw_min:=opc.popa_0082_cct_3242_b_raw_min;
//Map the analog scaling function block raw input to the physical raw input variable
cct_3242_b.raw_input := cct_3242_b_raw_input;

//Instantiate analog input function block
cct_3342_b();
//Map values from the OPC GVL so that they can be written to from outside POU(IE from HMI)
cct_3342_b.eu_max:=opc.popa_0082_cct_3342_b_eu_max;
cct_3342_b.eu_min:=opc.popa_0082_cct_3342_b_eu_min;
cct_3342_b.filter_factor:=opc.popa_0082_cct_3342_b_filter_factor;
cct_3342_b.raw_max:=opc.popa_0082_cct_3342_b_raw_max;
cct_3342_b.raw_min:=opc.popa_0082_cct_3342_b_raw_min;
//Map the analog scaling function block raw input to the physical raw input variable
cct_3342_b.raw_input := cct_3342_b_raw_input;

//Instantiate analog input function block
ft_3122_b();
//Map values from the OPC GVL so that they can be written to from outside POU(IE from HMI)
ft_3122_b.eu_max:=500;//opc.popa_0082_ft_3122_b_eu_max;
ft_3122_b.eu_min:=opc.popa_0082_ft_3122_b_eu_min;
ft_3122_b.filter_factor:=opc.popa_0082_ft_3122_b_filter_factor;
ft_3122_b.raw_max:=opc.popa_0082_ft_3122_b_raw_max;
ft_3122_b.raw_min:=opc.popa_0082_ft_3122_b_raw_min;
//Map the analog scaling function block raw input to the physical raw input variable
ft_3122_b.raw_input := ft_3122_b_raw_input;

//Instantiate analog input function block
ft_3222_b();
//Map values from the OPC GVL so that they can be written to from outside POU(IE from HMI)
ft_3222_b.eu_max:=500;//opc.popa_0082_ft_3222_b_eu_max;
ft_3222_b.eu_min:=opc.popa_0082_ft_3222_b_eu_min;
ft_3222_b.filter_factor:=opc.popa_0082_ft_3222_b_filter_factor;
ft_3222_b.raw_max:=opc.popa_0082_ft_3222_b_raw_max;
ft_3222_b.raw_min:=opc.popa_0082_ft_3222_b_raw_min;
//Map the analog scaling function block raw input to the physical raw input variable
ft_3222_b.raw_input := ft_3222_b_raw_input;

//Instantiate analog input function block
ft_3322_b();
//Map values from the OPC GVL so that they can be written to from outside POU(IE from HMI)
ft_3322_b.eu_max:=500;//opc.popa_0082_ft_3322_b_eu_max;
ft_3322_b.eu_min:=opc.popa_0082_ft_3322_b_eu_min;
ft_3322_b.filter_factor:=opc.popa_0082_ft_3322_b_filter_factor;
ft_3322_b.raw_max:=opc.popa_0082_ft_3322_b_raw_max;
ft_3322_b.raw_min:=opc.popa_0082_ft_3322_b_raw_min;
//Map the analog scaling function block raw input to the physical raw input variable
ft_3322_b.raw_input := ft_3322_b_raw_input;

//Instantiate analog input function block
lt_3102_b();
//Map values from the OPC GVL so that they can be written to from outside POU(IE from HMI)
lt_3102_b.eu_max:=opc.popa_0082_lt_3102_b_eu_max;
lt_3102_b.eu_min:=opc.popa_0082_lt_3102_b_eu_min;
lt_3102_b.filter_factor:=opc.popa_0082_lt_3102_b_filter_factor;
lt_3102_b.raw_max:=opc.popa_0082_lt_3102_b_raw_max;
lt_3102_b.raw_min:=opc.popa_0082_lt_3102_b_raw_min;
//Map the analog scaling function block raw input to the physical raw input variable
lt_3102_b.raw_input := lt_3102_b_raw_input;

//Instantiate analog input function block
lt_3202_b();
//Map values from the OPC GVL so that they can be written to from outside POU(IE from HMI)
lt_3202_b.eu_max:=opc.popa_0082_lt_3202_b_eu_max;
lt_3202_b.eu_min:=opc.popa_0082_lt_3202_b_eu_min;
lt_3202_b.filter_factor:=opc.popa_0082_lt_3202_b_filter_factor;
lt_3202_b.raw_max:=opc.popa_0082_lt_3202_b_raw_max;
lt_3202_b.raw_min:=opc.popa_0082_lt_3202_b_raw_min;
//Map the analog scaling function block raw input to the physical raw input variable
lt_3202_b.raw_input := lt_3202_b_raw_input;

//Instantiate analog input function block
lt_3302_b();
//Map values from the OPC GVL so that they can be written to from outside POU(IE from HMI)
lt_3302_b.eu_max:=opc.popa_0082_lt_3302_b_eu_max;
lt_3302_b.eu_min:=opc.popa_0082_lt_3302_b_eu_min;
lt_3302_b.filter_factor:=opc.popa_0082_lt_3302_b_filter_factor;
lt_3302_b.raw_max:=opc.popa_0082_lt_3302_b_raw_max;
lt_3302_b.raw_min:=opc.popa_0082_lt_3302_b_raw_min;
//Map the analog scaling function block raw input to the physical raw input variable
lt_3302_b.raw_input := lt_3302_b_raw_input;

//Instantiate analog input function block
lt_3153_b();
//Map values from the OPC GVL so that they can be written to from outside POU(IE from HMI)
lt_3153_b.eu_max:=opc.popa_0082_lt_3153_b_eu_max;
lt_3153_b.eu_min:=opc.popa_0082_lt_3153_b_eu_min;
lt_3153_b.filter_factor:=opc.popa_0082_lt_3153_b_filter_factor;
lt_3153_b.raw_max:=opc.popa_0082_lt_3153_b_raw_max;
lt_3153_b.raw_min:=opc.popa_0082_lt_3153_b_raw_min;
//Map the analog scaling function block raw input to the physical raw input variable
lt_3153_b.raw_input := lt_3153_b_raw_input;

//Instantiate analog input function block
lt_3253_b();
//Map values from the OPC GVL so that they can be written to from outside POU(IE from HMI)
lt_3253_b.eu_max:=opc.popa_0082_lt_3253_b_eu_max;
lt_3253_b.eu_min:=opc.popa_0082_lt_3253_b_eu_min;
lt_3253_b.filter_factor:=opc.popa_0082_lt_3253_b_filter_factor;
lt_3253_b.raw_max:=opc.popa_0082_lt_3253_b_raw_max;
lt_3253_b.raw_min:=opc.popa_0082_lt_3253_b_raw_min;
//Map the analog scaling function block raw input to the physical raw input variable
lt_3253_b.raw_input := lt_3253_b_raw_input;

//Instantiate analog input function block
lt_3353_b();
//Map values from the OPC GVL so that they can be written to from outside POU(IE from HMI)
lt_3353_b.eu_max:=opc.popa_0082_lt_3353_b_eu_max;
lt_3353_b.eu_min:=opc.popa_0082_lt_3353_b_eu_min;
lt_3353_b.filter_factor:=opc.popa_0082_lt_3353_b_filter_factor;
lt_3353_b.raw_max:=opc.popa_0082_lt_3353_b_raw_max;
lt_3353_b.raw_min:=opc.popa_0082_lt_3353_b_raw_min;
//Map the analog scaling function block raw input to the physical raw input variable
lt_3353_b.raw_input := lt_3353_b_raw_input;

//Instantiate analog input function block
lt_3402_b();
//Map values from the OPC GVL so that they can be written to from outside POU(IE from HMI)
lt_3402_b.eu_max:=opc.popa_0092_lt_3402_b_eu_max;
lt_3402_b.eu_min:=opc.popa_0092_lt_3402_b_eu_min;
lt_3402_b.filter_factor:=opc.popa_0092_lt_3402_b_filter_factor;
lt_3402_b.raw_max:=opc.popa_0092_lt_3402_b_raw_max;
lt_3402_b.raw_min:=opc.popa_0092_lt_3402_b_raw_min;
//Map the analog scaling function block raw input to the physical raw input variable
lt_3402_b.raw_input := lt_3402_b_raw_input;

//Instantiate analog input function block
pt_3119_b();
//Map values from the OPC GVL so that they can be written to from outside POU(IE from HMI)
pt_3119_b.eu_max:=opc.popa_0082_pt_3119_b_eu_max;
pt_3119_b.eu_min:=opc.popa_0082_pt_3119_b_eu_min;
pt_3119_b.filter_factor:=opc.popa_0082_pt_3119_b_filter_factor;
pt_3119_b.raw_max:=opc.popa_0082_pt_3119_b_raw_max;
pt_3119_b.raw_min:=opc.popa_0082_pt_3119_b_raw_min;
//Map the analog scaling function block raw input to the physical raw input variable
pt_3119_b.raw_input := pt_3119_b_raw_input;

//Instantiate analog input function block
pt_3219_b();
//Map values from the OPC GVL so that they can be written to from outside POU(IE from HMI)
pt_3219_b.eu_max:=opc.popa_0082_pt_3219_b_eu_max;
pt_3219_b.eu_min:=opc.popa_0082_pt_3219_b_eu_min;
pt_3219_b.filter_factor:=opc.popa_0082_pt_3219_b_filter_factor;
pt_3219_b.raw_max:=opc.popa_0082_pt_3219_b_raw_max;
pt_3219_b.raw_min:=opc.popa_0082_pt_3219_b_raw_min;
//Map the analog scaling function block raw input to the physical raw input variable
pt_3219_b.raw_input := pt_3219_b_raw_input;

//Instantiate analog input function block
pt_3319_b();
//Map values from the OPC GVL so that they can be written to from outside POU(IE from HMI)
pt_3319_b.eu_max:=opc.popa_0082_pt_3319_b_eu_max;
pt_3319_b.eu_min:=opc.popa_0082_pt_3319_b_eu_min;
pt_3319_b.filter_factor:=opc.popa_0082_pt_3319_b_filter_factor;
pt_3319_b.raw_max:=opc.popa_0082_pt_3319_b_raw_max;
pt_3319_b.raw_min:=opc.popa_0082_pt_3319_b_raw_min;
//Map the analog scaling function block raw input to the physical raw input variable
pt_3319_b.raw_input := pt_3319_b_raw_input;

//Instantiate analog input function block
pt_3141_b();
//Map values from the OPC GVL so that they can be written to from outside POU(IE from HMI)
pt_3141_b.eu_max:=opc.popa_0082_pt_3141_b_eu_max;
pt_3141_b.eu_min:=opc.popa_0082_pt_3141_b_eu_min;
pt_3141_b.filter_factor:=opc.popa_0082_pt_3141_b_filter_factor;
pt_3141_b.raw_max:=opc.popa_0082_pt_3141_b_raw_max;
pt_3141_b.raw_min:=opc.popa_0082_pt_3141_b_raw_min;
//Map the analog scaling function block raw input to the physical raw input variable
pt_3141_b.raw_input := pt_3141_b_raw_input;

//Instantiate analog input function block
pt_3241_b();
//Map values from the OPC GVL so that they can be written to from outside POU(IE from HMI)
pt_3241_b.eu_max:=opc.popa_0082_pt_3241_b_eu_max;
pt_3241_b.eu_min:=opc.popa_0082_pt_3241_b_eu_min;
pt_3241_b.filter_factor:=opc.popa_0082_pt_3241_b_filter_factor;
pt_3241_b.raw_max:=opc.popa_0082_pt_3241_b_raw_max;
pt_3241_b.raw_min:=opc.popa_0082_pt_3241_b_raw_min;
//Map the analog scaling function block raw input to the physical raw input variable
pt_3241_b.raw_input := pt_3241_b_raw_input;

//Instantiate analog input function block
pt_3341_b();
//Map values from the OPC GVL so that they can be written to from outside POU(IE from HMI)
pt_3341_b.eu_max:=opc.popa_0082_pt_3341_b_eu_max;
pt_3341_b.eu_min:=opc.popa_0082_pt_3341_b_eu_min;
pt_3341_b.filter_factor:=opc.popa_0082_pt_3341_b_filter_factor;
pt_3341_b.raw_max:=opc.popa_0082_pt_3341_b_raw_max;
pt_3341_b.raw_min:=opc.popa_0082_pt_3341_b_raw_min;
//Map the analog scaling function block raw input to the physical raw input variable
pt_3341_b.raw_input := pt_3341_b_raw_input;

//Instantiate analog input function block
pt_3428_b();
//Map values from the OPC GVL so that they can be written to from outside POU(IE from HMI)
pt_3428_b.eu_max:=opc.popa_0092_pt_3428_b_eu_max;
pt_3428_b.eu_min:=opc.popa_0092_pt_3428_b_eu_min;
pt_3428_b.filter_factor:=opc.popa_0092_pt_3428_b_filter_factor;
pt_3428_b.raw_max:=opc.popa_0092_pt_3428_b_raw_max;
pt_3428_b.raw_min:=opc.popa_0092_pt_3428_b_raw_min;
//Map the analog scaling function block raw input to the physical raw input variable
pt_3428_b.raw_input := pt_3428_b_raw_input;

//Instantiate analog input function block
pt_3414_b();
//Map values from the OPC GVL so that they can be written to from outside POU(IE from HMI)
pt_3414_b.eu_max:=opc.popa_0092_pt_3414_b_eu_max;
pt_3414_b.eu_min:=opc.popa_0092_pt_3414_b_eu_min;
pt_3414_b.filter_factor:=opc.popa_0092_pt_3414_b_filter_factor;
pt_3414_b.raw_max:=opc.popa_0092_pt_3414_b_raw_max;
pt_3414_b.raw_min:=opc.popa_0092_pt_3414_b_raw_min;
//Map the analog scaling function block raw input to the physical raw input variable
pt_3414_b.raw_input := pt_3414_b_raw_input;

//Instantiate analog input function block
tt_3118_b();
//Map values from the OPC GVL so that they can be written to from outside POU(IE from HMI)
tt_3118_b.eu_max:=opc.popa_0082_tt_3118_b_eu_max;
tt_3118_b.eu_min:=opc.popa_0082_tt_3118_b_eu_min;
tt_3118_b.filter_factor:=opc.popa_0082_tt_3118_b_filter_factor;
tt_3118_b.raw_max:=opc.popa_0082_tt_3118_b_raw_max;
tt_3118_b.raw_min:=opc.popa_0082_tt_3118_b_raw_min;
//Map the analog scaling function block raw input to the physical raw input variable
tt_3118_b.raw_input := tt_3118_b_raw_input;

//Instantiate analog input function block
tt_3218_b();
//Map values from the OPC GVL so that they can be written to from outside POU(IE from HMI)
tt_3218_b.eu_max:=opc.popa_0082_tt_3218_b_eu_max;
tt_3218_b.eu_min:=opc.popa_0082_tt_3218_b_eu_min;
tt_3218_b.filter_factor:=opc.popa_0082_tt_3218_b_filter_factor;
tt_3218_b.raw_max:=opc.popa_0082_tt_3218_b_raw_max;
tt_3218_b.raw_min:=opc.popa_0082_tt_3218_b_raw_min;
//Map the analog scaling function block raw input to the physical raw input variable
tt_3218_b.raw_input := tt_3218_b_raw_input;

//Instantiate analog input function block
tt_3318_b();
//Map values from the OPC GVL so that they can be written to from outside POU(IE from HMI)
tt_3318_b.eu_max:=opc.popa_0082_tt_3318_b_eu_max;
tt_3318_b.eu_min:=opc.popa_0082_tt_3318_b_eu_min;
tt_3318_b.filter_factor:=opc.popa_0082_tt_3318_b_filter_factor;
tt_3318_b.raw_max:=opc.popa_0082_tt_3318_b_raw_max;
tt_3318_b.raw_min:=opc.popa_0082_tt_3318_b_raw_min;
//Map the analog scaling function block raw input to the physical raw input variable
tt_3318_b.raw_input := tt_3318_b_raw_input;

//Instantiate analog input function block
tt_3140_b();
//Map values from the OPC GVL so that they can be written to from outside POU(IE from HMI)
tt_3140_b.eu_max:=opc.popa_0082_tt_3140_b_eu_max;
tt_3140_b.eu_min:=opc.popa_0082_tt_3140_b_eu_min;
tt_3140_b.filter_factor:=opc.popa_0082_tt_3140_b_filter_factor;
tt_3140_b.raw_max:=opc.popa_0082_tt_3140_b_raw_max;
tt_3140_b.raw_min:=opc.popa_0082_tt_3140_b_raw_min;
//Map the analog scaling function block raw input to the physical raw input variable
tt_3140_b.raw_input := tt_3140_b_raw_input;

//Instantiate analog input function block
tt_3240_b();
//Map values from the OPC GVL so that they can be written to from outside POU(IE from HMI)
tt_3240_b.eu_max:=opc.popa_0082_tt_3240_b_eu_max;
tt_3240_b.eu_min:=opc.popa_0082_tt_3240_b_eu_min;
tt_3240_b.filter_factor:=opc.popa_0082_tt_3240_b_filter_factor;
tt_3240_b.raw_max:=opc.popa_0082_tt_3240_b_raw_max;
tt_3240_b.raw_min:=opc.popa_0082_tt_3240_b_raw_min;
//Map the analog scaling function block raw input to the physical raw input variable
tt_3240_b.raw_input := tt_3240_b_raw_input;

//Instantiate analog input function block
tt_3340_b();
//Map values from the OPC GVL so that they can be written to from outside POU(IE from HMI)
tt_3340_b.eu_max:=opc.popa_0082_tt_3340_b_eu_max;
tt_3340_b.eu_min:=opc.popa_0082_tt_3340_b_eu_min;
tt_3340_b.filter_factor:=opc.popa_0082_tt_3340_b_filter_factor;
tt_3340_b.raw_max:=opc.popa_0082_tt_3340_b_raw_max;
tt_3340_b.raw_min:=opc.popa_0082_tt_3340_b_raw_min;
//Map the analog scaling function block raw input to the physical raw input variable
tt_3340_b.raw_input := tt_3340_b_raw_input;

//Instantiate analog input function block
tt_3432_b();
//Map values from the OPC GVL so that they can be written to from outside POU(IE from HMI)
tt_3432_b.eu_max:=opc.popa_0092_tt_3432_b_eu_max;
tt_3432_b.eu_min:=opc.popa_0092_tt_3432_b_eu_min;
tt_3432_b.filter_factor:=opc.popa_0092_tt_3432_b_filter_factor;
tt_3432_b.raw_max:=opc.popa_0092_tt_3432_b_raw_max;
tt_3432_b.raw_min:=opc.popa_0092_tt_3432_b_raw_min;
//Map the analog scaling function block raw input to the physical raw input variable
tt_3432_b.raw_input := tt_3432_b_raw_input;

//---Pumps---------------------------------------------------------------------------------------------------------------------------------



//Instantiate u_3112_b speed feedback analog input function block
u_3112_b_speed_feedback();
//Map values from the OPC GVL so that they can be written to from outside POU(IE from HMI)
u_3112_b_speed_feedback.eu_max:=60;
u_3112_b_speed_feedback.eu_min:=0;
u_3112_b_speed_feedback.filter_factor:=opc.popa_0082_u_3112_b_speed_feedback_filter_factor;
u_3112_b_speed_feedback.raw_max:=opc.popa_0082_u_3112_b_speed_feedback_raw_max;
u_3112_b_speed_feedback.raw_min:=opc.popa_0082_u_3112_b_speed_feedback_raw_min;
//Map the analog scaling function block raw input to the physical raw input variable
u_3112_b_speed_feedback.raw_input := u_3112_b_speed_feedback_raw_input;





//--------------------------------------------------------------------------------------------------------------


//Instantiate Example analog input function block
u_3212_b_speed_feedback();
//Map values from the OPC GVL so that they can be written to from outside POU(IE from HMI)
u_3212_b_speed_feedback.eu_max:=60;
u_3212_b_speed_feedback.eu_min:=0;
u_3212_b_speed_feedback.filter_factor:=opc.popa_0082_u_3212_b_speed_feedback_filter_factor;
u_3212_b_speed_feedback.raw_max:=opc.popa_0082_u_3212_b_speed_feedback_raw_max;
u_3212_b_speed_feedback.raw_min:=opc.popa_0082_u_3212_b_speed_feedback_raw_min;
//Map the analog scaling function block raw input to the physical raw input variable
u_3212_b_speed_feedback.raw_input := u_3212_b_speed_feedback_raw_input;

//--------------------------------------------------------------------------------------------------------------


//Instantiate Example analog input function block
u_3312_b_speed_feedback();
//Map values from the OPC GVL so that they can be written to from outside POU(IE from HMI)
u_3312_b_speed_feedback.eu_max:=60;
u_3312_b_speed_feedback.eu_min:=0;
u_3312_b_speed_feedback.filter_factor:=opc.popa_0082_u_3312_b_speed_feedback_filter_factor;
u_3312_b_speed_feedback.raw_max:=opc.popa_0082_u_3312_b_speed_feedback_raw_max;
u_3312_b_speed_feedback.raw_min:=opc.popa_0082_u_3312_b_speed_feedback_raw_min;
//Map the analog scaling function block raw input to the physical raw input variable
u_3312_b_speed_feedback.raw_input := u_3312_b_speed_feedback_raw_input;

//--------------------------------------------------------------------------------------------------------------


//Instantiate Example analog input function block
u_3160_b_speed_feedback();
//Map values from the OPC GVL so that they can be written to from outside POU(IE from HMI)
u_3160_b_speed_feedback.eu_max:=60;
u_3160_b_speed_feedback.eu_min:=0;
u_3160_b_speed_feedback.filter_factor:=opc.popa_0082_u_3160_b_speed_feedback_filter_factor;
u_3160_b_speed_feedback.raw_max:=opc.popa_0082_u_3160_b_speed_feedback_raw_max;
u_3160_b_speed_feedback.raw_min:=opc.popa_0082_u_3160_b_speed_feedback_raw_min;
//Map the analog scaling function block raw input to the physical raw input variable
u_3160_b_speed_feedback.raw_input := u_3160_b_speed_feedback_raw_input;

//--------------------------------------------------------------------------------------------------------------


//Instantiate Example analog input function block
u_3260_b_speed_feedback();
//Map values from the OPC GVL so that they can be written to from outside POU(IE from HMI)
u_3260_b_speed_feedback.eu_max:=60;
u_3260_b_speed_feedback.eu_min:=0;
u_3260_b_speed_feedback.filter_factor:=opc.popa_0082_u_3260_b_speed_feedback_filter_factor;
u_3260_b_speed_feedback.raw_max:=opc.popa_0082_u_3260_b_speed_feedback_raw_max;
u_3260_b_speed_feedback.raw_min:=opc.popa_0082_u_3260_b_speed_feedback_raw_min;
//Map the analog scaling function block raw input to the physical raw input variable
u_3260_b_speed_feedback.raw_input := u_3260_b_speed_feedback_raw_input;

//--------------------------------------------------------------------------------------------------------------


//Instantiate Example analog input function block
u_3360_b_speed_feedback();
//Map values from the OPC GVL so that they can be written to from outside POU(IE from HMI)
u_3360_b_speed_feedback.eu_max:=60;
u_3360_b_speed_feedback.eu_min:=0;
u_3360_b_speed_feedback.filter_factor:=opc.popa_0082_u_3360_b_speed_feedback_filter_factor;
u_3360_b_speed_feedback.raw_max:=opc.popa_0082_u_3360_b_speed_feedback_raw_max;
u_3360_b_speed_feedback.raw_min:=opc.popa_0082_u_3360_b_speed_feedback_raw_min;
//Map the analog scaling function block raw input to the physical raw input variable
u_3360_b_speed_feedback.raw_input := u_3360_b_speed_feedback_raw_input;

//--------------------------------------------------------------------------------------------------------------


//Instantiate Example analog input function block
u_3370_b_speed_feedback();
//Map values from the OPC GVL so that they can be written to from outside POU(IE from HMI)
u_3370_b_speed_feedback.eu_max:=60;
u_3370_b_speed_feedback.eu_min:=0;
u_3370_b_speed_feedback.filter_factor:=opc.popa_0082_u_3370_b_speed_feedback_filter_factor;
u_3370_b_speed_feedback.raw_max:=opc.popa_0082_u_3370_b_speed_feedback_raw_max;
u_3370_b_speed_feedback.raw_min:=opc.popa_0082_u_3370_b_speed_feedback_raw_min;
//Map the analog scaling function block raw input to the physical raw input variable
u_3370_b_speed_feedback.raw_input := u_3370_b_speed_feedback_raw_input;

//--------------------------------------------------------------------------------------------------------------


//Instantiate Example analog input function block
u_3405_b_speed_feedback();
//Map values from the OPC GVL so that they can be written to from outside POU(IE from HMI)
u_3405_b_speed_feedback.eu_max:=60;
u_3405_b_speed_feedback.eu_min:=0;
u_3405_b_speed_feedback.filter_factor:=opc.popa_0092_u_3405_b_speed_feedback_filter_factor;
u_3405_b_speed_feedback.raw_max:=opc.popa_0092_u_3405_b_speed_feedback_raw_max;
u_3405_b_speed_feedback.raw_min:=opc.popa_0092_u_3405_b_speed_feedback_raw_min;
//Map the analog scaling function block raw input to the physical raw input variable
u_3405_b_speed_feedback.raw_input := u_3405_b_speed_feedback_raw_input;


//---Valves----------------------------------------------------------------------------------------------------------------------------------------------

//Instantiate av_3148 analog input function block----------------------------------------------------------------------------
av_3148_b_position_feedback();
//Map values from the OPC GVL so that they can be written to from outside POU(IE from HMI)
av_3148_b_position_feedback.eu_max:=100;
av_3148_b_position_feedback.eu_min:=0;
av_3148_b_position_feedback.filter_factor:=opc.popa_0082_av_3148_b_position_feedback_filter_factor;
av_3148_b_position_feedback.raw_max:=opc.popa_0082_av_3148_b_position_feedback_raw_max;
av_3148_b_position_feedback.raw_min:=opc.popa_0082_av_3148_b_position_feedback_raw_min;
//Map the analog scaling function block raw input to the physical raw input variable
av_3148_b_position_feedback.raw_input := av_3148_b_position_feedback_raw_input;




//Instantiate av_3248 analog input function block-----------------------------------------------------------------
av_3248_b_position_feedback();
//Map values from the OPC GVL so that they can be written to from outside POU(IE from HMI)
av_3248_b_position_feedback.eu_max:=100;
av_3248_b_position_feedback.eu_min:=0;
av_3248_b_position_feedback.filter_factor:=opc.popa_0082_av_3248_b_position_feedback_filter_factor;
av_3248_b_position_feedback.raw_max:=opc.popa_0082_av_3248_b_position_feedback_raw_max;
av_3248_b_position_feedback.raw_min:=opc.popa_0082_av_3248_b_position_feedback_raw_min;
//Map the analog scaling function block raw input to the physical raw input variable
av_3248_b_position_feedback.raw_input := av_3248_b_position_feedback_raw_input;




//Instantiate av_3348 analog input function block----------------------------------------------------------------------
av_3348_b_position_feedback();
//Map values from the OPC GVL so that they can be written to from outside POU(IE from HMI)
av_3348_b_position_feedback.eu_max:=100;
av_3348_b_position_feedback.eu_min:=0;
av_3348_b_position_feedback.filter_factor:=opc.popa_0082_av_3348_b_position_feedback_filter_factor;
av_3348_b_position_feedback.raw_max:=opc.popa_0082_av_3348_b_position_feedback_raw_max;
av_3348_b_position_feedback.raw_min:=opc.popa_0082_av_3348_b_position_feedback_raw_min;
//Map the analog scaling function block raw input to the physical raw input variable
av_3348_b_position_feedback.raw_input := av_3348_b_position_feedback_raw_input;

END_PROGRAM

// ---- POUs/manual_mode.TcPOU
PROGRAM manual_mode
VAR
	//manual_mode: BOOL;
	
	u_3112_a_hmi_start_request: BOOL;
	u_3112_a_manual_request: BOOL;
	u_3112_a_hmi_speed_request: REAL;
	u_3112_a_manual_speed_request: REAL;
	u_3112_a_hmi_stop_request: BOOL;
	
	u_3212_a_hmi_start_request: BOOL;
	u_3212_a_manual_request: BOOL;
	u_3212_a_hmi_speed_request: REAL;
	u_3212_a_manual_speed_request: REAL;
	u_3212_a_hmi_stop_request: BOOL;

	u_3312_a_hmi_start_request: BOOL;
	u_3312_a_manual_request: BOOL;
	u_3312_a_hmi_speed_request: REAL;
	u_3312_a_manual_speed_request: REAL;
	u_3312_a_hmi_stop_request: BOOL;
	
	u_3405_a_hmi_start_request: BOOL;
	u_3405_a_manual_request: BOOL;
	u_3405_a_hmi_speed_request: REAL;
	u_3405_a_manual_speed_request: REAL;
	u_3405_a_hmi_stop_request: BOOL;
	
	u_3160_a_hmi_start_request: BOOL;
	u_3160_a_manual_request: BOOL;
	u_3160_a_hmi_speed_request: REAL;
	u_3160_a_manual_speed_request: REAL;
	u_3160_a_hmi_stop_request: BOOL;
	
	u_3260_a_hmi_start_request: BOOL;
	u_3260_a_manual_request: BOOL;
	u_3260_a_hmi_speed_request: REAL;
	u_3260_a_manual_speed_request: REAL;
	u_3260_a_hmi_stop_request: BOOL;
	
	u_3360_a_hmi_start_request: BOOL;
	u_3360_a_manual_request: BOOL;
	u_3360_a_hmi_speed_request: REAL;
	u_3360_a_manual_speed_request: REAL;
	u_3360_a_hmi_stop_request: BOOL;
	
	nv_3110_a_hmi_open_request: BOOL;
	nv_3110_a_hmi_close_request: BOOL;
	nv_3110_a_manual_request: BOOL;
	
	nv_3210_a_hmi_open_request: BOOL;
	nv_3210_a_hmi_close_request: BOOL;
	nv_3210_a_manual_request: BOOL;
	
	nv_3310_a_hmi_open_request: BOOL;
	nv_3310_a_hmi_close_request: BOOL;
	nv_3310_a_manual_request: BOOL;
	
	nv_3135_a_hmi_open_request: BOOL;
	nv_3135_a_hmi_close_request: BOOL;
	nv_3135_a_manual_request: BOOL;
	
	nv_3235_a_hmi_open_request: BOOL;
	nv_3235_a_hmi_close_request: BOOL;
	nv_3235_a_manual_request: BOOL;
	
	nv_3335_a_hmi_open_request: BOOL;
	nv_3335_a_hmi_close_request: BOOL;
	nv_3335_a_manual_request: BOOL;
	
	nv_3372_a_hmi_open_request: BOOL;
	nv_3372_a_hmi_close_request: BOOL;
	nv_3372_a_manual_request: BOOL;
	u_3370_a_hmi_start_request: BOOL;
	u_3370_a_manual_request: BOOL;
	u_3370_a_hmi_stop_request: BOOL;
	u_3370_a_hmi_speed_request: INT;
	u_3370_a_manual_speed_request: INT;
	nv_3162_a_hmi_open_request: BOOL;
	nv_3162_a_manual_request: BOOL;
	nv_3162_a_hmi_close_request: BOOL;
END_VAR

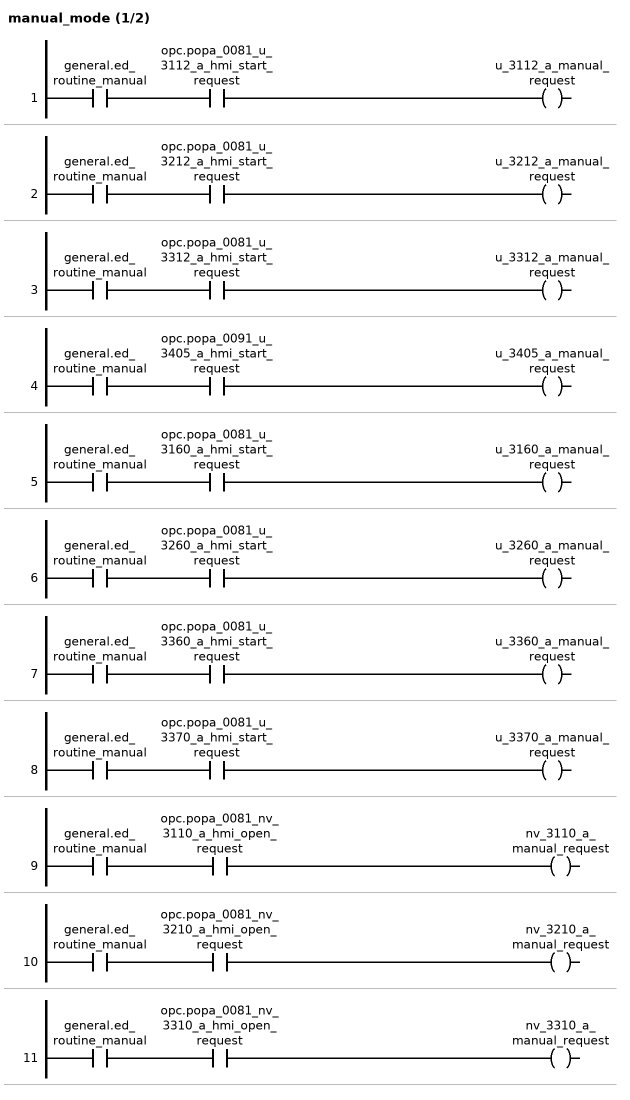
// NETWORK 1
u_3112_a_manual_request := general.ed_routine_manual AND opc.popa_0081_u_3112_a_hmi_start_request;

// NETWORK 2
u_3212_a_manual_request := general.ed_routine_manual AND opc.popa_0081_u_3212_a_hmi_start_request;

// NETWORK 3
u_3312_a_manual_request := general.ed_routine_manual AND opc.popa_0081_u_3312_a_hmi_start_request;

// NETWORK 4
u_3405_a_manual_request := general.ed_routine_manual AND opc.popa_0091_u_3405_a_hmi_start_request;

// NETWORK 5
u_3160_a_manual_request := general.ed_routine_manual AND opc.popa_0081_u_3160_a_hmi_start_request;

// NETWORK 6
u_3260_a_manual_request := general.ed_routine_manual AND opc.popa_0081_u_3260_a_hmi_start_request;

// NETWORK 7
u_3360_a_manual_request := general.ed_routine_manual AND opc.popa_0081_u_3360_a_hmi_start_request;

// NETWORK 8
u_3370_a_manual_request := general.ed_routine_manual AND opc.popa_0081_u_3370_a_hmi_start_request;

// NETWORK 9
nv_3110_a_manual_request := general.ed_routine_manual AND opc.popa_0081_nv_3110_a_hmi_open_request;

// NETWORK 10
nv_3210_a_manual_request := general.ed_routine_manual AND opc.popa_0081_nv_3210_a_hmi_open_request;

// NETWORK 11
nv_3310_a_manual_request := general.ed_routine_manual AND opc.popa_0081_nv_3310_a_hmi_open_request;

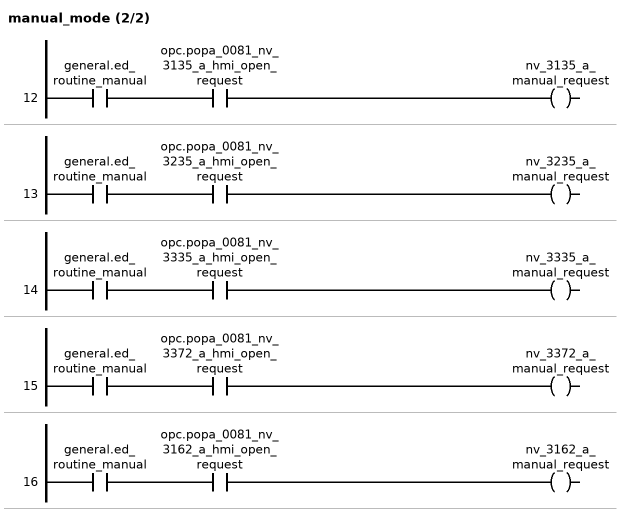
// NETWORK 12
nv_3135_a_manual_request := general.ed_routine_manual AND opc.popa_0081_nv_3135_a_hmi_open_request;

// NETWORK 13
nv_3235_a_manual_request := general.ed_routine_manual AND opc.popa_0081_nv_3235_a_hmi_open_request;

// NETWORK 14
nv_3335_a_manual_request := general.ed_routine_manual AND opc.popa_0081_nv_3335_a_hmi_open_request;

// NETWORK 15
nv_3372_a_manual_request := general.ed_routine_manual AND opc.popa_0081_nv_3372_a_hmi_open_request;

// NETWORK 16
nv_3162_a_manual_request := general.ed_routine_manual AND opc.popa_0081_nv_3162_a_hmi_open_request;

END_PROGRAM

// ---- POUs/interlocks.TcPOU
PROGRAM interlocks
VAR PERSISTENT
	nv_3110_a_open: BOOL;
	alm_lt_3012_a_low: BOOL;
	intlk_u3112: BOOL;
	nv_3210_a_open: BOOL;
	nv_3310_a_open: BOOL;
	intlk_u3212: BOOL;
	intlk_u3312: BOOL;
	alm_lt_3102_a_low: BOOL;
	alm_lt_3202_a_low: BOOL;
	alm_lt_3302_a_low: BOOL;
	alm_lt_3153_a_low: BOOL;
	intlk_u3160: BOOL;
	alm_lt_3253_a_low: BOOL;
	intlk_u3260: BOOL;
	alm_lt_3353_a_low: BOOL;
	intlk_u3360: BOOL;
	nv_3372_a_open: BOOL;
	intlk_u3370: BOOL;
	alm_lt_3402_a_low: BOOL;
	nv_3135_a_open: BOOL;
	nv_3235_a_open: BOOL;
	nv_3335: BOOL;
	nv_3335_a_open: BOOL;
	intlk_nv3110: BOOL;
	u_3112_a_running: BOOL;
END_VAR

VAR
	intlk_nv3210: BOOL;
	u_3212_a_running: BOOL;
	intlk_nv3310: BOOL;
	u_3312_a_running: BOOL;
	u_3112_a_intlk: BOOL;
	nv_3110_a_intlk: BOOL;
	u_3212_a_intlk: BOOL;
	nv_3210_a_intlk: BOOL;
	u_3312_a_intlk: BOOL;
	nv_3310_a_intlk: BOOL;
	u_3160_a_intlk: BOOL;
	u_3260_a_intlk: BOOL;
	u_3360_a_intlk: BOOL;
	u_3370_a_intlk: BOOL;
	u_3405_a_intlk: BOOL;
END_VAR

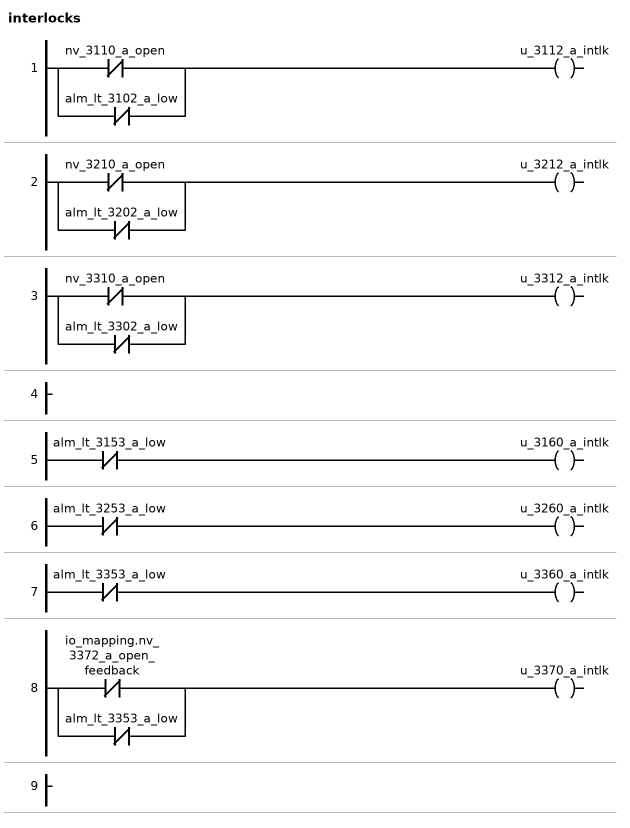
// NETWORK 1
u_3112_a_intlk := NOT nv_3110_a_open OR NOT alm_lt_3102_a_low;

// NETWORK 2
u_3212_a_intlk := NOT nv_3210_a_open OR NOT alm_lt_3202_a_low;

// NETWORK 3
u_3312_a_intlk := NOT nv_3310_a_open OR NOT alm_lt_3302_a_low;

// NETWORK 4

// NETWORK 5
u_3160_a_intlk := NOT alm_lt_3153_a_low;

// NETWORK 6
u_3260_a_intlk := NOT alm_lt_3253_a_low;

// NETWORK 7
u_3360_a_intlk := NOT alm_lt_3353_a_low;

// NETWORK 8
u_3370_a_intlk := NOT io_mapping.nv_3372_a_open_feedback OR NOT alm_lt_3353_a_low;

// NETWORK 9

END_PROGRAM

// ---- POUs/maint_mode.TcPOU
PROGRAM maint_mode
VAR
	maint_mode: BOOL;
	
	u_3112_b_hmi_start_request: BOOL;
	u_3112_b_maint_request: BOOL;
	u_3112_b_hmi_speed_request: REAL;
	u_3112_b_maint_speed_request: REAL;
	u_3112_b_hmi_stop_request: BOOL;
	
	u_3212_b_hmi_start_request: BOOL;
	u_3212_b_maint_request: BOOL;
	u_3212_b_hmi_speed_request: REAL;
	u_3212_b_maint_speed_request: REAL;
	u_3212_b_hmi_stop_request: BOOL;

	u_3312_b_hmi_start_request: BOOL;
	u_3312_b_maint_request: BOOL;
	u_3312_b_hmi_speed_request: REAL;
	u_3312_b_maint_speed_request: REAL;
	u_3312_b_hmi_stop_request: BOOL;
	
	u_3405_b_hmi_start_request: BOOL;
	u_3405_b_maint_request: BOOL;
	u_3405_b_hmi_speed_request: REAL;
	u_3405_b_maint_speed_request: REAL;
	u_3405_b_hmi_stop_request: BOOL;
	
	u_3160_b_hmi_start_request: BOOL;
	u_3160_b_maint_request: BOOL;
	u_3160_b_hmi_speed_request: REAL;
	u_3160_b_maint_speed_request: REAL;
	u_3160_b_hmi_stop_request: BOOL;
	
	u_3260_b_hmi_start_request: BOOL;
	u_3260_b_maint_request: BOOL;
	u_3260_b_hmi_speed_request: REAL;
	u_3260_b_maint_speed_request: REAL;
	u_3260_b_hmi_stop_request: BOOL;
	
	u_3360_b_hmi_start_request: BOOL;
	u_3360_b_maint_request: BOOL;
	u_3360_b_hmi_speed_request: REAL;
	u_3360_b_maint_speed_request: REAL;
	u_3360_b_hmi_stop_request: BOOL;
	
	nv_3110_b_hmi_open_request: BOOL;
	nv_3110_b_hmi_close_request: BOOL;
	nv_3110_b_maint_request: BOOL;
	
	nv_3210_b_hmi_open_request: BOOL;
	nv_3210_b_hmi_close_request: BOOL;
	nv_3210_b_maint_request: BOOL;
	
	nv_3310_b_hmi_open_request: BOOL;
	nv_3310_b_hmi_close_request: BOOL;
	nv_3310_b_maint_request: BOOL;
	
	nv_3135_b_hmi_open_request: BOOL;
	nv_3135_b_hmi_close_request: BOOL;
	nv_3135_b_maint_request: BOOL;
	
	nv_3235_b_hmi_open_request: BOOL;
	nv_3235_b_hmi_close_request: BOOL;
	nv_3235_b_maint_request: BOOL;
	
	nv_3335_b_hmi_open_request: BOOL;
	nv_3335_b_hmi_close_request: BOOL;
	nv_3335_b_maint_request: BOOL;
	
	nv_3372_b_hmi_open_request: BOOL;
	nv_3372_b_hmi_close_request: BOOL;
	nv_3372_b_maint_request: BOOL;
	u_3370_b_hmi_start_request: BOOL;
	u_3370_b_maint_request: BOOL;
	u_3370_b_hmi_stop_request: BOOL;
	u_3370_b_hmi_speed_request: REAL;
	u_3370_b_maint_speed_request: REAL;
	nv_3162_b_hmi_open_request: BOOL;
	nv_3162_b_maint_request: BOOL;
	nv_3162_b_hmi_close_request: BOOL;
END_VAR

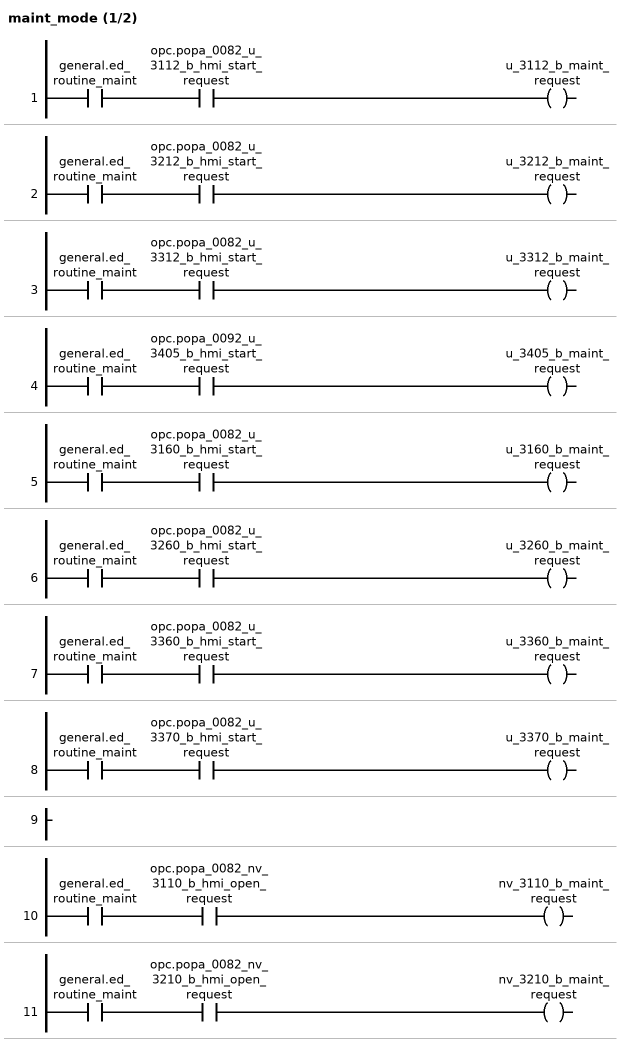
// NETWORK 1
u_3112_b_maint_request := general.ed_routine_maint AND opc.popa_0082_u_3112_b_hmi_start_request;

// NETWORK 2
u_3212_b_maint_request := general.ed_routine_maint AND opc.popa_0082_u_3212_b_hmi_start_request;

// NETWORK 3
u_3312_b_maint_request := general.ed_routine_maint AND opc.popa_0082_u_3312_b_hmi_start_request;

// NETWORK 4
u_3405_b_maint_request := general.ed_routine_maint AND opc.popa_0092_u_3405_b_hmi_start_request;

// NETWORK 5
u_3160_b_maint_request := general.ed_routine_maint AND opc.popa_0082_u_3160_b_hmi_start_request;

// NETWORK 6
u_3260_b_maint_request := general.ed_routine_maint AND opc.popa_0082_u_3260_b_hmi_start_request;

// NETWORK 7
u_3360_b_maint_request := general.ed_routine_maint AND opc.popa_0082_u_3360_b_hmi_start_request;

// NETWORK 8
u_3370_b_maint_request := general.ed_routine_maint AND opc.popa_0082_u_3370_b_hmi_start_request;

// NETWORK 9

// NETWORK 10
nv_3110_b_maint_request := general.ed_routine_maint AND opc.popa_0082_nv_3110_b_hmi_open_request;

// NETWORK 11
nv_3210_b_maint_request := general.ed_routine_maint AND opc.popa_0082_nv_3210_b_hmi_open_request;

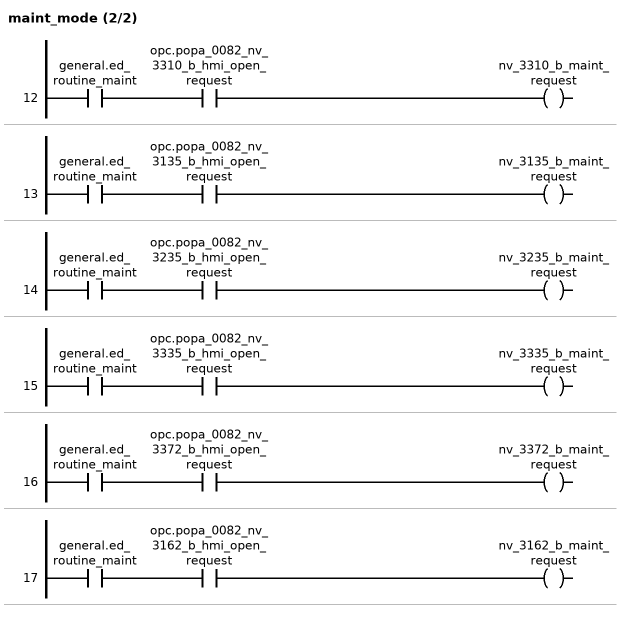
// NETWORK 12
nv_3310_b_maint_request := general.ed_routine_maint AND opc.popa_0082_nv_3310_b_hmi_open_request;

// NETWORK 13
nv_3135_b_maint_request := general.ed_routine_maint AND opc.popa_0082_nv_3135_b_hmi_open_request;

// NETWORK 14
nv_3235_b_maint_request := general.ed_routine_maint AND opc.popa_0082_nv_3235_b_hmi_open_request;

// NETWORK 15
nv_3335_b_maint_request := general.ed_routine_maint AND opc.popa_0082_nv_3335_b_hmi_open_request;

// NETWORK 16
nv_3372_b_maint_request := general.ed_routine_maint AND opc.popa_0082_nv_3372_b_hmi_open_request;

// NETWORK 17
nv_3162_b_maint_request := general.ed_routine_maint AND opc.popa_0082_nv_3162_b_hmi_open_request;

END_PROGRAM

// ---- POUs/stopping_mode.TcPOU
PROGRAM stopping_mode
VAR
	ed_routine_stopping_idle: BOOL;
	stack_power_enabled: BOOL;
	RECTIFIER_OUTPUT_OFF: BOOL;// ADD LOGIC FOR MONITORING RECTIFIER OUTPUT - USE CT? VERIFY PS DOES NOT MOVE CURRENT WHEN POWERED OFF
	u_3112_b_stop_request: BOOL;
	u_3212_b_stop_request: BOOL;
	u_3312_b_stop_request: BOOL;
	u_3405_b_stop_request: BOOL;
	u_3160_b_stop_request: BOOL
;
	u_3260_b_stop_request: BOOL;
	u_3360_b_stop_request: BOOL;
	u_3370_b_stop_request: BOOL;
	u_3112_b_run_feedback: BOOL;
	u_3212_b_run_feedback: BOOL;
	u_3312_b_run_feedback: BOOL;
	u_3405_b_run_feedback: BOOL;
	u_3160_b_run_feedback: BOOL;
	u_3260_b_run_feedback: BOOL;
	u_3360_b_run_feedback: BOOL;
	u_3370_b_run_feedback: BOOL;
	
	nv_3110_b_stop_request:BOOL;
	av_3248_b_stop_request: BOOL;
	av_3148_b_stop_request: BOOL;
	nv_3335_b_stop_request: BOOL;
	nv_3235_b_stop_request: BOOL;
	nv_3135_b_stop_request: BOOL;
	nv_3310_b_stop_request: BOOL;
	nv_3210_b_stop_request: BOOL;
	ed_routine_stop_mode: BOOL;
	redox_doser_stop_request: BOOL;
	nv_3335_b_position_request: INT;
	av_3148_b_position_request: INT;
	av_3248_b_position_request: INT;
	ed_pumps_stopped: BOOL;

	nv_3335_b_position_feedback: INT;
	nv_3335_b_recycle_position: BOOL;
	av_3148_b_position_feedback: INT;
	av_3148_b_recycle_position: BOOL;
	av_3248_b_recycle_position: BOOL;
	ed_valves_stopped: BOOL;
	ed_stopped: BOOL;
	av_3348_b_position_request: INT;
	nv_3372_b_stop_request: BOOL;
	av_3348_b_position_feedback: INT;
	av_3348_b_recycle_position: BOOL;
	nv_3335_b_closed_feedback: BOOL;
	nv_3372_b_closed_feedback: BOOL;
	nv_3162_b_stop_request: BOOL;
	ed_critical_stop: BOOL;
	tmr_stop_pump_delay: TON;
	tmr_stop_pump_delay_pt: TIME := T#10S;
	tmr_stop_pump_delay_et: TIME;
	test_ramp: ramp;
	eng_test: BOOL;
	test_ramp_start_val: REAL;
	test_ramp_end_val: REAL;
	test_ramp_duration: INT;
END_VAR
VAR // added by the converter: edge detectors and wires of the graphical bodies
    _w1, _w2, _w3 : BOOL;
END_VAR

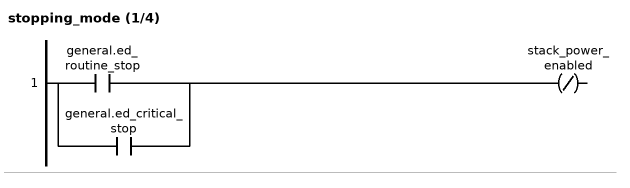
// NETWORK 1
stack_power_enabled := NOT (general.ed_routine_stop OR general.ed_critical_stop);

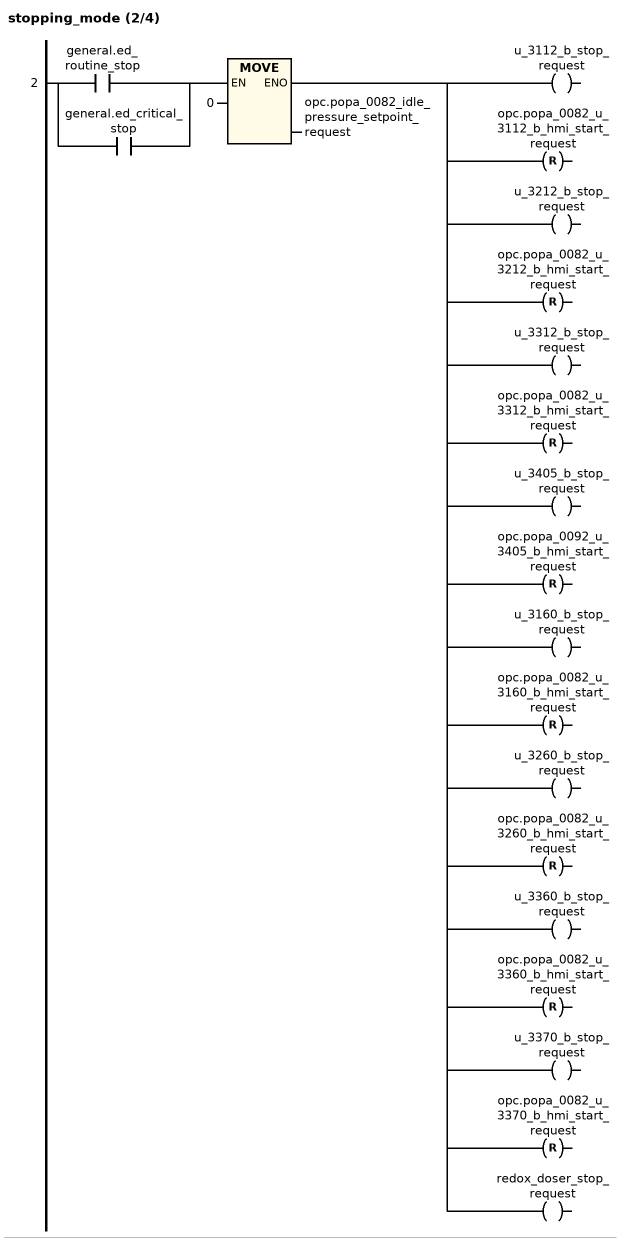
// NETWORK 2
_w1 := general.ed_routine_stop OR general.ed_critical_stop;
IF _w1 THEN opc.popa_0082_idle_pressure_setpoint_request := 0; END_IF
u_3112_b_stop_request := _w1;
opc.popa_0082_u_3112_b_hmi_start_request R= _w1;
u_3212_b_stop_request := _w1;
opc.popa_0082_u_3212_b_hmi_start_request R= _w1;
u_3312_b_stop_request := _w1;
opc.popa_0082_u_3312_b_hmi_start_request R= _w1;
u_3405_b_stop_request := _w1;
opc.popa_0092_u_3405_b_hmi_start_request R= _w1;
u_3160_b_stop_request := _w1;
opc.popa_0082_u_3160_b_hmi_start_request R= _w1;
u_3260_b_stop_request := _w1;
opc.popa_0082_u_3260_b_hmi_start_request R= _w1;
u_3360_b_stop_request := _w1;
opc.popa_0082_u_3360_b_hmi_start_request R= _w1;
u_3370_b_stop_request := _w1;
opc.popa_0082_u_3370_b_hmi_start_request R= _w1;
redox_doser_stop_request := _w1;

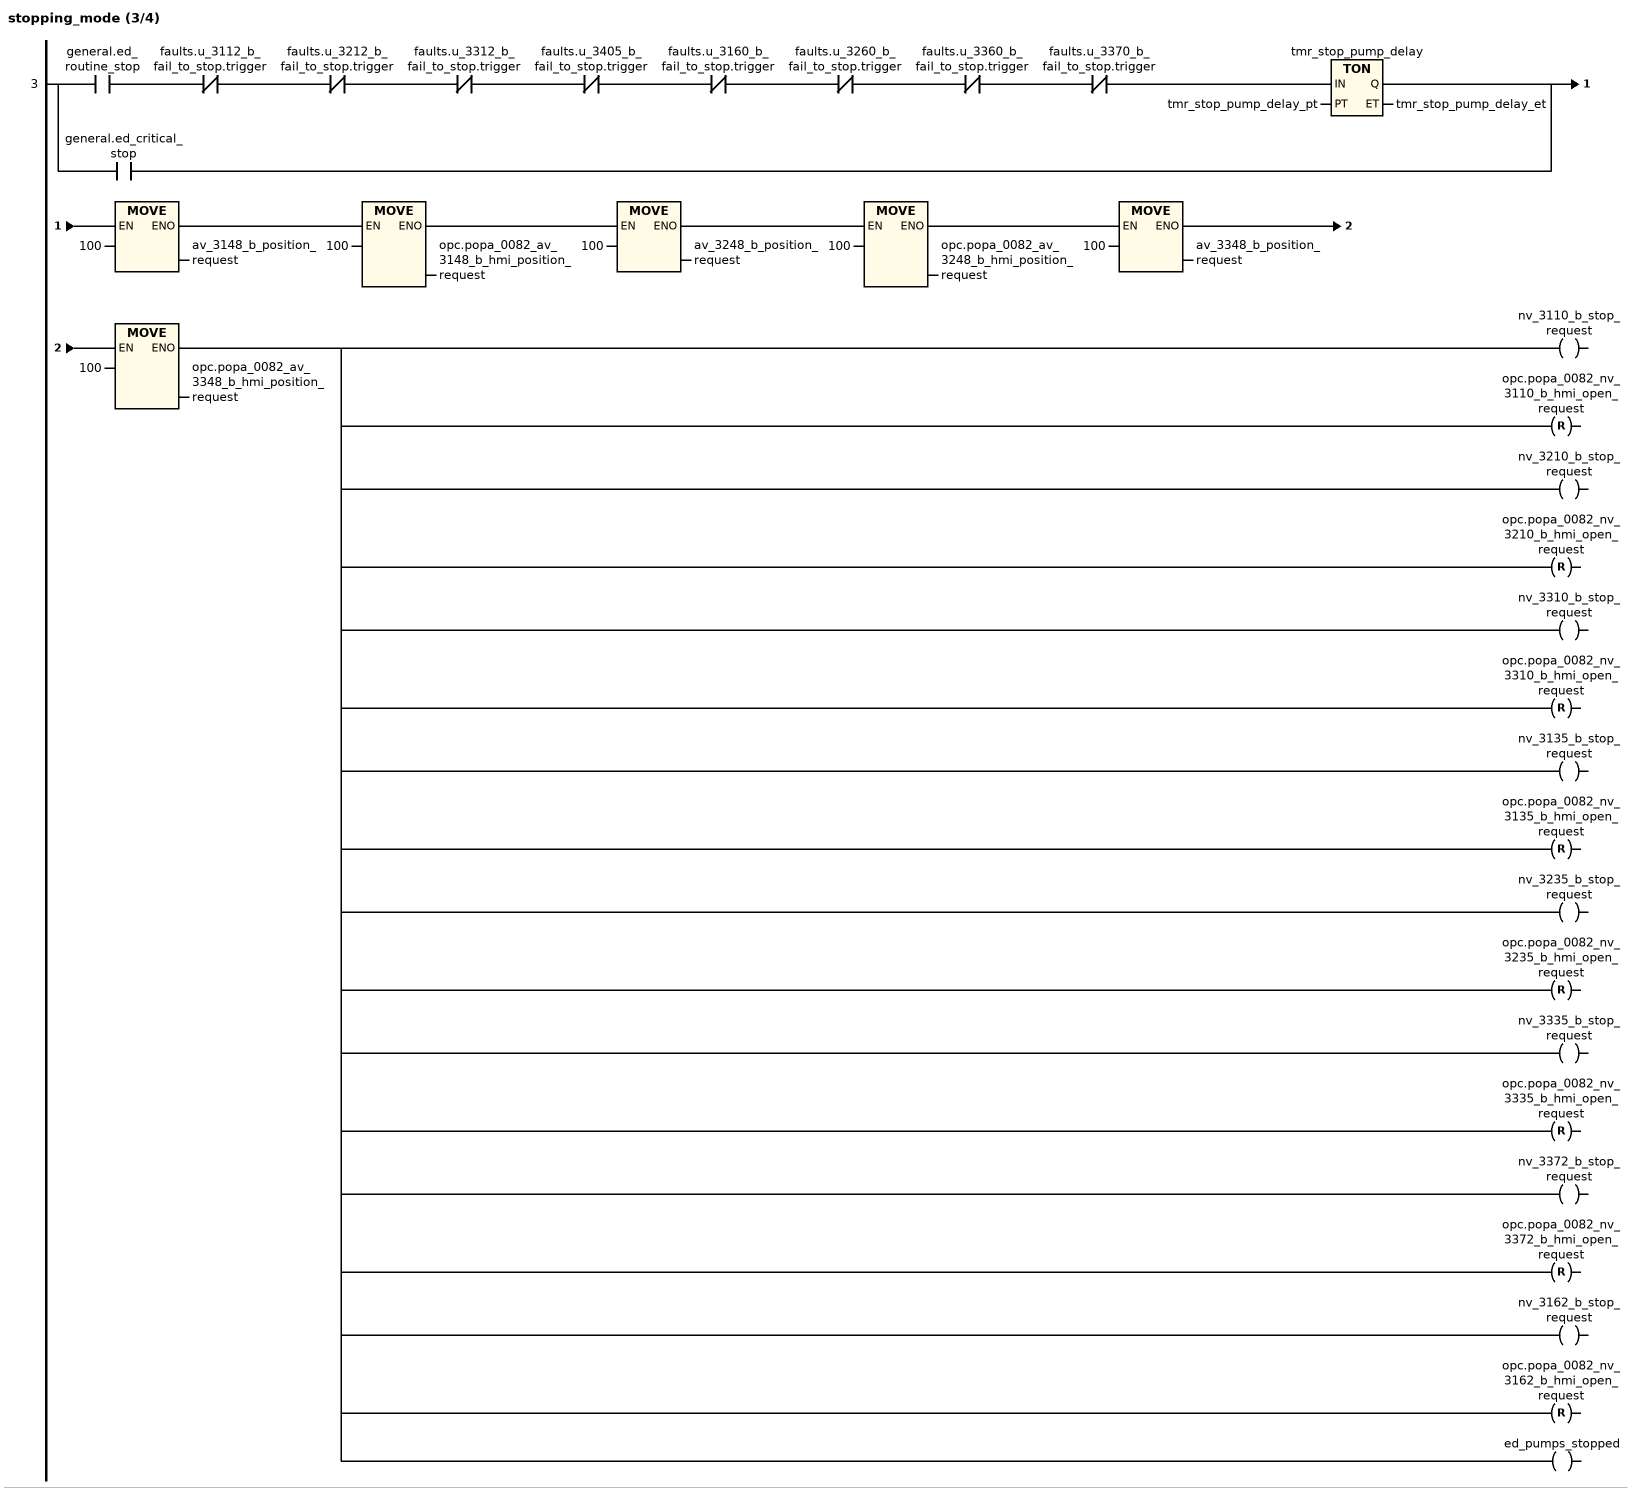
// NETWORK 3
tmr_stop_pump_delay(
    IN := general.ed_routine_stop AND NOT faults.u_3112_b_fail_to_stop.trigger AND NOT faults.u_3212_b_fail_to_stop.trigger AND NOT faults.u_3312_b_fail_to_stop.trigger AND NOT faults.u_3405_b_fail_to_stop.trigger AND NOT faults.u_3160_b_fail_to_stop.trigger AND NOT faults.u_3260_b_fail_to_stop.trigger AND NOT faults.u_3360_b_fail_to_stop.trigger AND NOT faults.u_3370_b_fail_to_stop.trigger,
    PT := tmr_stop_pump_delay_pt,
    ET => tmr_stop_pump_delay_et); // TON
_w2 := tmr_stop_pump_delay.Q OR general.ed_critical_stop;
IF _w2 THEN av_3148_b_position_request := 100; END_IF
IF _w2 THEN opc.popa_0082_av_3148_b_hmi_position_request := 100; END_IF
IF _w2 THEN av_3248_b_position_request := 100; END_IF
IF _w2 THEN opc.popa_0082_av_3248_b_hmi_position_request := 100; END_IF
IF _w2 THEN av_3348_b_position_request := 100; END_IF
IF _w2 THEN opc.popa_0082_av_3348_b_hmi_position_request := 100; END_IF
nv_3110_b_stop_request := _w2;
opc.popa_0082_nv_3110_b_hmi_open_request R= _w2;
nv_3210_b_stop_request := _w2;
opc.popa_0082_nv_3210_b_hmi_open_request R= _w2;
nv_3310_b_stop_request := _w2;
opc.popa_0082_nv_3310_b_hmi_open_request R= _w2;
nv_3135_b_stop_request := _w2;
opc.popa_0082_nv_3135_b_hmi_open_request R= _w2;
nv_3235_b_stop_request := _w2;
opc.popa_0082_nv_3235_b_hmi_open_request R= _w2;
nv_3335_b_stop_request := _w2;
opc.popa_0082_nv_3335_b_hmi_open_request R= _w2;
nv_3372_b_stop_request := _w2;
opc.popa_0082_nv_3372_b_hmi_open_request R= _w2;
nv_3162_b_stop_request := _w2;
opc.popa_0082_nv_3162_b_hmi_open_request R= _w2;
ed_pumps_stopped := _w2;

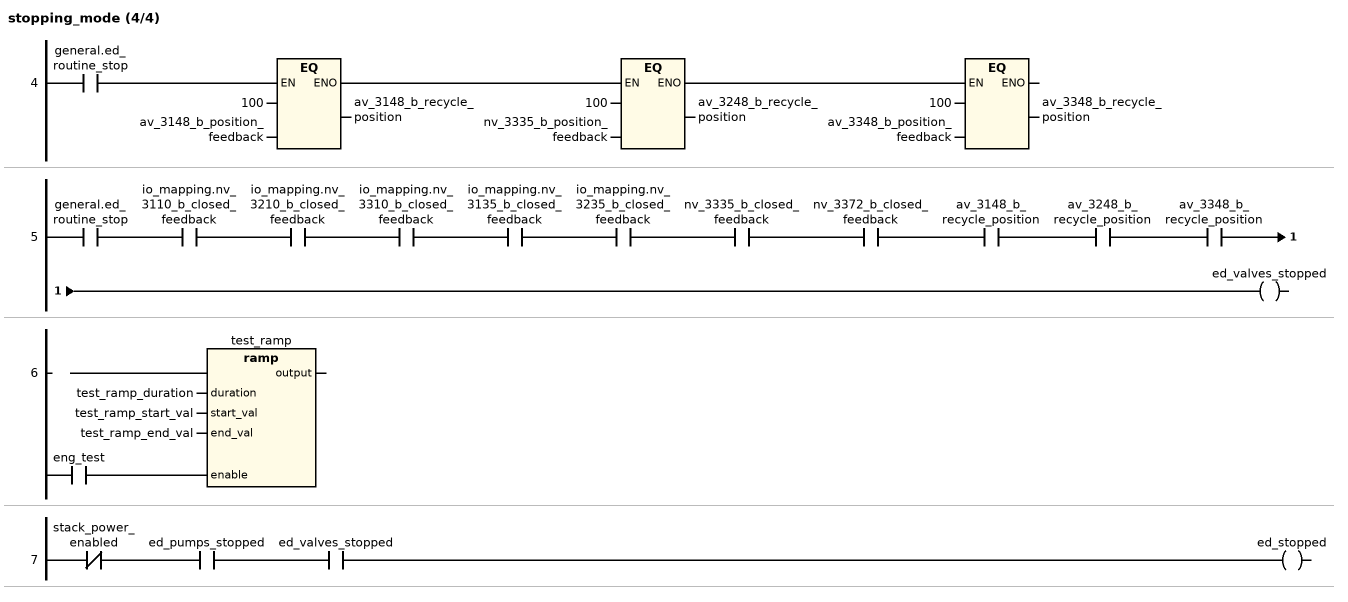
// NETWORK 4
_w3 := general.ed_routine_stop;
IF _w3 THEN av_3148_b_recycle_position := 100 = av_3148_b_position_feedback; END_IF
IF _w3 THEN av_3248_b_recycle_position := 100 = nv_3335_b_position_feedback; END_IF
IF _w3 THEN av_3348_b_recycle_position := 100 = av_3348_b_position_feedback; END_IF

// NETWORK 5
ed_valves_stopped := general.ed_routine_stop AND io_mapping.nv_3110_b_closed_feedback AND io_mapping.nv_3210_b_closed_feedback AND io_mapping.nv_3310_b_closed_feedback AND io_mapping.nv_3135_b_closed_feedback AND io_mapping.nv_3235_b_closed_feedback AND nv_3335_b_closed_feedback AND nv_3372_b_closed_feedback AND av_3148_b_recycle_position AND av_3248_b_recycle_position AND av_3348_b_recycle_position;

// NETWORK 6
test_ramp(
    duration := test_ramp_duration,
    start_val := test_ramp_start_val,
    end_val := test_ramp_end_val,
    enable := eng_test); // ramp

// NETWORK 7
ed_stopped := NOT stack_power_enabled AND ed_pumps_stopped AND ed_valves_stopped;

END_PROGRAM

// ---- POUs/cip.TcPOU
PROGRAM cip
VAR
	ed_routine_starting_idle: BOOL;
	idle_redox_doser_enable: BOOL;
	
	tmr_idle_pumps: TON;
	idle_u_3112_b_request: BOOL;
	idle_u_3312_b_request: BOOL;
	idle_u_3405_b_request: BOOL;
	idle_u_3212_b_request: BOOL;
	tmr_idle_pump_delay: TON;
	u_3112_b_running: BOOL;
	u_3112_b_speed_ref: INT;
	u_3112_b_sp: REAL;
	salt_pressure_actual: REAL;
	idle_u_3112_b_ready: BOOL;
	u_3212_b_running: BOOL;
	idle_u_3212_b_ready: BOOL;
	idle_u_3312_b_ready: BOOL;
	u_3312_b_running: BOOL;
	u_3405_b_running: BOOL;
	idle_u_3405_b_ready: BOOL;
	idle_stack_power_enable: BOOL;
	ed_routine_cip: BOOL;
	
		nv_3110_b_open_request: BOOL;
	nv_3210_b_open_request: BOOL;
	nv_3310_b_open_request: BOOL;
	nv_3110_b_open_feedback: BOOL;
	nv_3210_b_open_feedback: BOOL;
	nv_3310_b_open_feedback: BOOL;
	cip_redox_doser_enable: BOOL;
	nv_3372_b_open_request: BOOL;
	nv_3135_b_open_request: BOOL;
	nv_3235_b_open_request: BOOL;
	nv_3335_b_open_request: BOOL;
	nv_3372_b_open_feedback: BOOL;
	nv_3135_b_open_feedback: BOOL;
	nv_3235_b_open_feedback: BOOL;
	nv_3335_b_open_feedback: BOOL;
	tmr_cip_pump_delay: TON;
	idle_u_3370_b_request: BOOL;
	u_3370_b_running: BOOL;
	u_3370_b_sp: REAL;
	tmr_cip_pump_start_delay: TON;
	tmr_cip_run: TON;
	cip_tmr_preset: TIME;
	
	u_3370_b_actual: INT; // What would this be???
	ft_3122_b_tot: INT;
	ft_3222_b_tot: INT;
	ft_3322_b_tot: INT;
	cip_flush_tot: INT;
	cip_flush_sp: INT;
	cip_u_3370_b_request: BOOL;
	cip_complete: BOOL;
	cip_stop_request: BOOL;
	nv_3372_b_cip_request: BOOL;
	nv_3135_b_cip_request: BOOL;
	nv_3235_b_cip_request: BOOL;
	nv_3335_b_cip_request: BOOL;
	redox_doser_cip_enable: BOOL;
	u_3370_b_cip_request: BOOL;
	CIP_TEMP_BIT: BOOL;
	tmr_cip_valve_delay: TON;
	tmr_cip_valve_delay_pt: TIME:= T#30S;
	tmr_cip_valve_delay_et: TIME;
	tmr_cip_valve_delay_q: BOOL;
	u_3112_b_cip_pressure_setpoint_request: REAL;
	u_3370_b_cip_pressure_setpoint_request: REAL;
END_VAR
VAR // added by the converter: edge detectors and wires of the graphical bodies
    _w1, _w2, _w3 : BOOL;
END_VAR

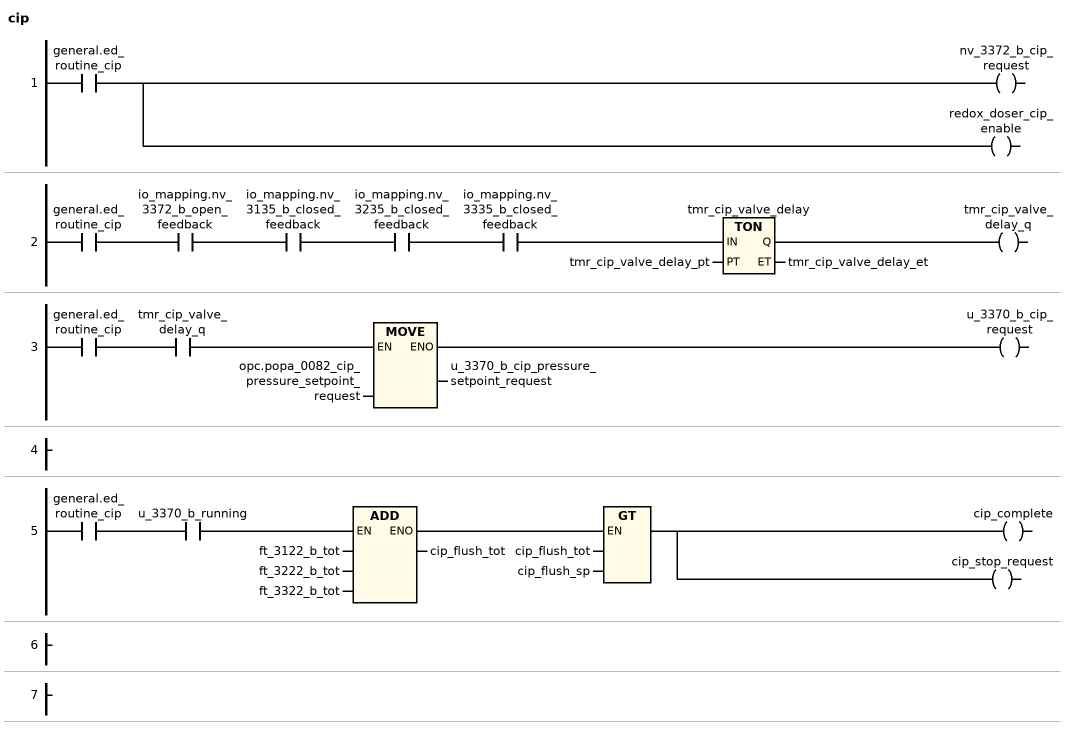
// NETWORK 1
nv_3372_b_cip_request := general.ed_routine_cip;
redox_doser_cip_enable := general.ed_routine_cip;

// NETWORK 2
tmr_cip_valve_delay(
    IN := general.ed_routine_cip AND io_mapping.nv_3372_b_open_feedback AND io_mapping.nv_3135_b_closed_feedback AND io_mapping.nv_3235_b_closed_feedback AND io_mapping.nv_3335_b_closed_feedback,
    PT := tmr_cip_valve_delay_pt,
    ET => tmr_cip_valve_delay_et); // TON
tmr_cip_valve_delay_q := tmr_cip_valve_delay.Q;

// NETWORK 3
_w1 := general.ed_routine_cip AND tmr_cip_valve_delay_q;
IF _w1 THEN u_3370_b_cip_pressure_setpoint_request := opc.popa_0082_cip_pressure_setpoint_request; END_IF
u_3370_b_cip_request := _w1;

// NETWORK 4

// NETWORK 5
_w2 := general.ed_routine_cip AND u_3370_b_running;
IF _w2 THEN cip_flush_tot := ft_3122_b_tot + ft_3222_b_tot + ft_3322_b_tot; END_IF
_w3 := _w2 AND cip_flush_tot > cip_flush_sp;
cip_complete := _w3;
cip_stop_request := _w3;

// NETWORK 6

// NETWORK 7

END_PROGRAM

// ---- POUs/valve_manager.TcPOU
PROGRAM valve_manager
VAR
	//Digital valve
	nv_3110_a: valve_digital;
	nv_3210_a: valve_digital;
	nv_3310_a: valve_digital;
	nv_3135_a: valve_digital;
	nv_3235_a: valve_digital;
	nv_3335_a: valve_digital;
	nv_3372_a: valve_digital;
	nv_3162_a: valve_digital;
	
	// Analog Valve Function Block
	av_3148_a: valve_analog;
	av_3248_a: valve_analog;
	av_3348_a: valve_analog;


	//Repeat for each valve?
	u_3112_a_open_request: BOOL;
	u_3112_a_idle_request: BOOL;
	u_3112_a_cip_request: BOOL;
	u_3112_a_manual_request: BOOL;
	u_3112_a_stop_request: BOOL;
	u_3112_a_intlk: BOOL;
	gen_alm_active: BOOL;
	ed_routine_idle: BOOL;
	ed_routine_cip: BOOL;
	ed_routine_manual: BOOL;
	ed_routine_maint: BOOL;
	nv_3110_a_idle_request: BOOL;
	nv_3110_a_cip_request: BOOL;
	nv_3110_a_manual_request: BOOL;
	nv_3110_a_intlk: BOOL;
	nv_3110_a_stop_request: BOOL;
	nv_3110_a_open_request: BOOL;
	nv_3210_a_open_request: BOOL;
	nv_3310_a_open_request: BOOL;
	nv_3135_a_open_request: BOOL;
	nv_3235_a_open_request: BOOL;
	nv_3335_a_open_request: BOOL;
	nv_3372_a_open_request: BOOL;
	nv_3210_a_idle_request: BOOL;
	nv_3210_a_cip_request: BOOL;
	nv_3210_a_manual_request: BOOL;
	nv_3210_a_stop_request: BOOL;
	nv_3210_a_intlk: BOOL;
	
	nv_3310_a_idle_request: BOOL;
	nv_3310_a_cip_request: BOOL;
	nv_3310_a_manual_request: BOOL;
	nv_3310_a_stop_request: BOOL;
	nv_3310_a_intlk: BOOL;
	
	nv_3135_a_idle_request: BOOL;
	nv_3135_a_cip_request: BOOL;
	nv_3135_a_manual_request: BOOL;
	nv_3135_a_stop_request: BOOL;
	nv_3135_a_intlk: BOOL;
	
	nv_3235_a_idle_request: BOOL;
	nv_3235_a_cip_request: BOOL;
	nv_3235_a_manual_request: BOOL;
	nv_3235_a_stop_request: BOOL;
	nv_3235_a_intlk: BOOL;
	
	nv_3335_a_idle_request: BOOL;
	nv_3335_a_cip_request: BOOL;
	nv_3335_a_manual_request: BOOL;
	nv_3335_a_stop_request: BOOL;
	nv_3335_a_intlk: BOOL;
	
	nv_3372_a_idle_request: BOOL;
	nv_3372_a_cip_request: BOOL;
	nv_3372_a_manual_request: BOOL;
	nv_3372_a_stop_request: BOOL;
	nv_3372_a_intlk: BOOL;
	
	nv_3162_a_idle_request: BOOL;
	nv_3162_a_cip_request: BOOL;
	nv_3162_a_manual_request: BOOL;
	nv_3162_a_stop_request: BOOL;
	nv_3162_a_intlk: BOOL;
	nv_3162_a_open_request: BOOL;
	
	av_3148_a_idle_request: BOOL;
	av_3148_a_cip_request: BOOL;
	av_3148_a_idle_position_request: REAL;
	av_3148_a_position_request: REAL;
	av_3148_a_cip_position_request: REAL;
	av_3148_a_manual_position_request: REAL;
	av_3148_a_manual_request: BOOL;
	av_3148_a_maint_request: BOOL;
	av_3148_a_maint_position_request: REAL;
	av_3148_a_intlk: BOOL;
	av_3148_a_stop_request: BOOL;
	av_3148_a_open_request: BOOL;
	
	av_3248_a_idle_request: BOOL;
	av_3248_a_cip_request: BOOL;
	av_3248_a_idle_position_request: REAL;
	av_3248_a_position_request: REAL;
	av_3248_a_cip_position_request: REAL;
	av_3248_a_manual_position_request: REAL;
	av_3248_a_manual_request: BOOL;
	av_3248_a_maint_request: BOOL;
	av_3248_a_maint_position_request: REAL;
	av_3248_a_intlk: BOOL;
	av_3248_a_stop_request: BOOL;
	av_3248_a_open_request: BOOL;
	
	av_3348_a_idle_request: BOOL;
	av_3348_a_cip_request: BOOL;
	av_3348_a_idle_position_request: REAL;
	av_3348_a_position_request: REAL;
	av_3348_a_cip_position_request: REAL;
	av_3348_a_manual_position_request: REAL;
	av_3348_a_manual_request: BOOL;
	av_3348_a_maint_request: BOOL;
	av_3348_a_maint_position_request: REAL;
	av_3348_a_intlk: BOOL;
	av_3348_a_stop_request: BOOL;
	av_3348_a_open_request: BOOL;
	
END_VAR
VAR // added by the converter: edge detectors and wires of the graphical bodies
    _w1, _w2, _w3, _w4, _w5, _w6, _w7, _w8, _w9, _w10, _w11, _w12, _w13, _w14, _w15 : BOOL;
END_VAR

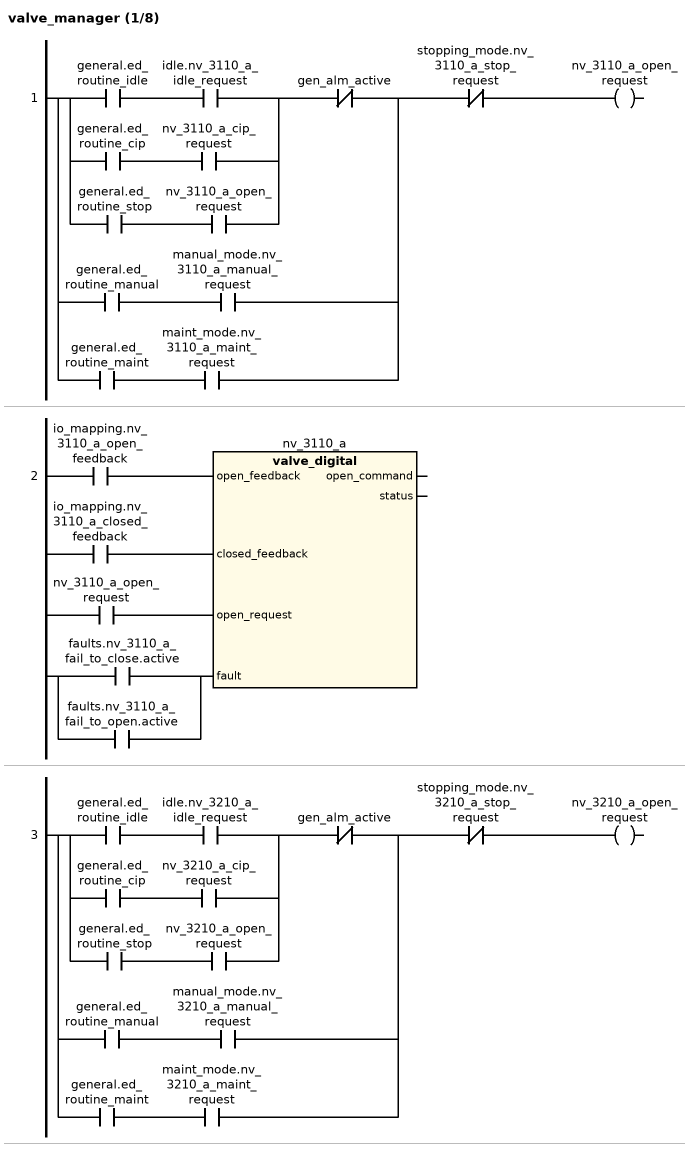
// NETWORK 1
nv_3110_a_open_request := ((general.ed_routine_idle AND idle.nv_3110_a_idle_request OR general.ed_routine_cip AND nv_3110_a_cip_request OR general.ed_routine_stop AND nv_3110_a_open_request) AND NOT gen_alm_active OR general.ed_routine_manual AND manual_mode.nv_3110_a_manual_request OR general.ed_routine_maint AND maint_mode.nv_3110_a_maint_request) AND NOT stopping_mode.nv_3110_a_stop_request;

// NETWORK 2
nv_3110_a(
    open_feedback := io_mapping.nv_3110_a_open_feedback,
    closed_feedback := io_mapping.nv_3110_a_closed_feedback,
    open_request := nv_3110_a_open_request,
    fault := faults.nv_3110_a_fail_to_close.active OR faults.nv_3110_a_fail_to_open.active); // valve_digital

// NETWORK 3
nv_3210_a_open_request := ((general.ed_routine_idle AND idle.nv_3210_a_idle_request OR general.ed_routine_cip AND nv_3210_a_cip_request OR general.ed_routine_stop AND nv_3210_a_open_request) AND NOT gen_alm_active OR general.ed_routine_manual AND manual_mode.nv_3210_a_manual_request OR general.ed_routine_maint AND maint_mode.nv_3210_a_maint_request) AND NOT stopping_mode.nv_3210_a_stop_request;

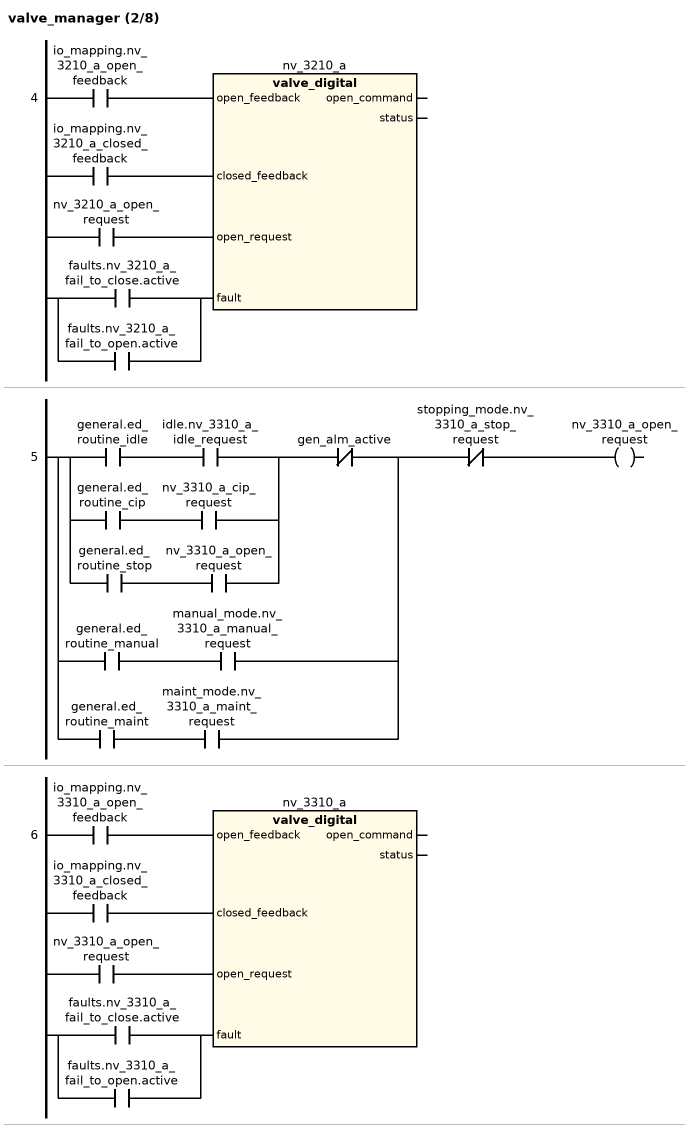
// NETWORK 4
nv_3210_a(
    open_feedback := io_mapping.nv_3210_a_open_feedback,
    closed_feedback := io_mapping.nv_3210_a_closed_feedback,
    open_request := nv_3210_a_open_request,
    fault := faults.nv_3210_a_fail_to_close.active OR faults.nv_3210_a_fail_to_open.active); // valve_digital

// NETWORK 5
nv_3310_a_open_request := ((general.ed_routine_idle AND idle.nv_3310_a_idle_request OR general.ed_routine_cip AND nv_3310_a_cip_request OR general.ed_routine_stop AND nv_3310_a_open_request) AND NOT gen_alm_active OR general.ed_routine_manual AND manual_mode.nv_3310_a_manual_request OR general.ed_routine_maint AND maint_mode.nv_3310_a_maint_request) AND NOT stopping_mode.nv_3310_a_stop_request;

// NETWORK 6
nv_3310_a(
    open_feedback := io_mapping.nv_3310_a_open_feedback,
    closed_feedback := io_mapping.nv_3310_a_closed_feedback,
    open_request := nv_3310_a_open_request,
    fault := faults.nv_3310_a_fail_to_close.active OR faults.nv_3310_a_fail_to_open.active); // valve_digital

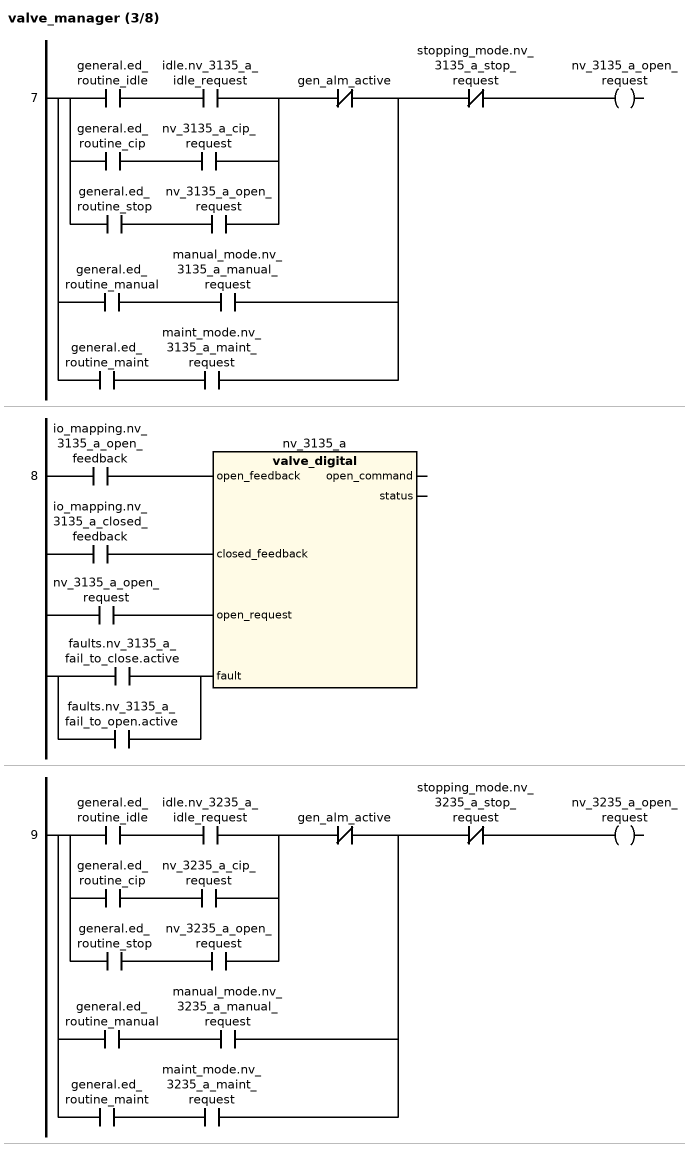
// NETWORK 7
nv_3135_a_open_request := ((general.ed_routine_idle AND idle.nv_3135_a_idle_request OR general.ed_routine_cip AND nv_3135_a_cip_request OR general.ed_routine_stop AND nv_3135_a_open_request) AND NOT gen_alm_active OR general.ed_routine_manual AND manual_mode.nv_3135_a_manual_request OR general.ed_routine_maint AND maint_mode.nv_3135_a_maint_request) AND NOT stopping_mode.nv_3135_a_stop_request;

// NETWORK 8
nv_3135_a(
    open_feedback := io_mapping.nv_3135_a_open_feedback,
    closed_feedback := io_mapping.nv_3135_a_closed_feedback,
    open_request := nv_3135_a_open_request,
    fault := faults.nv_3135_a_fail_to_close.active OR faults.nv_3135_a_fail_to_open.active); // valve_digital

// NETWORK 9
nv_3235_a_open_request := ((general.ed_routine_idle AND idle.nv_3235_a_idle_request OR general.ed_routine_cip AND nv_3235_a_cip_request OR general.ed_routine_stop AND nv_3235_a_open_request) AND NOT gen_alm_active OR general.ed_routine_manual AND manual_mode.nv_3235_a_manual_request OR general.ed_routine_maint AND maint_mode.nv_3235_a_maint_request) AND NOT stopping_mode.nv_3235_a_stop_request;

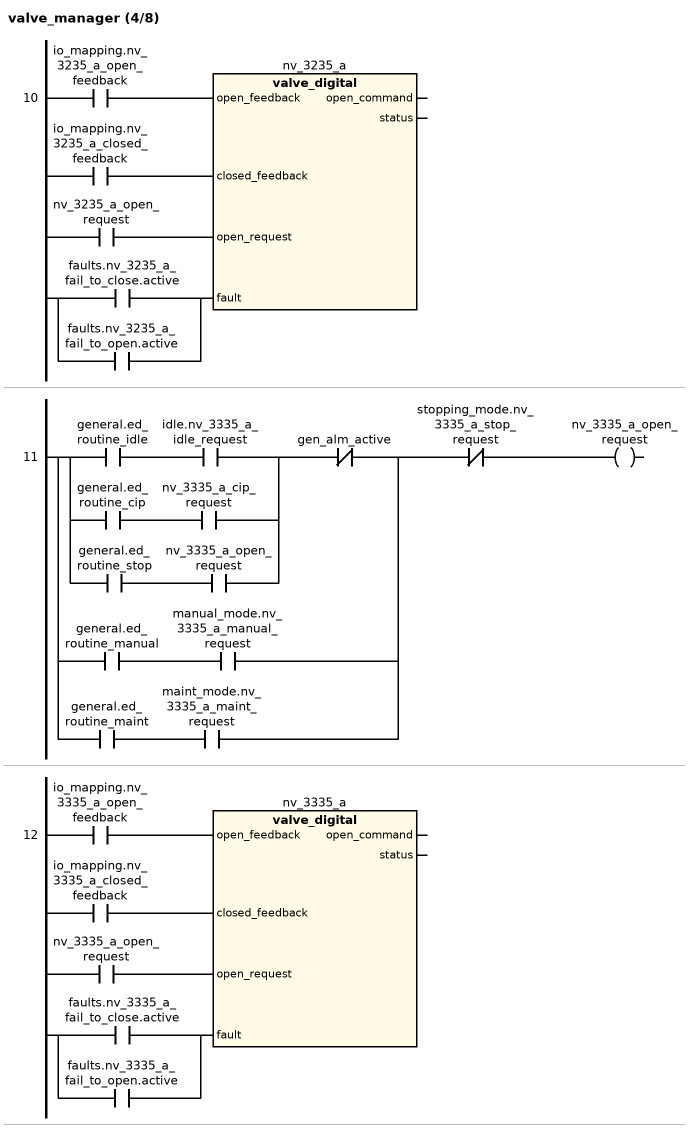
// NETWORK 10
nv_3235_a(
    open_feedback := io_mapping.nv_3235_a_open_feedback,
    closed_feedback := io_mapping.nv_3235_a_closed_feedback,
    open_request := nv_3235_a_open_request,
    fault := faults.nv_3235_a_fail_to_close.active OR faults.nv_3235_a_fail_to_open.active); // valve_digital

// NETWORK 11
nv_3335_a_open_request := ((general.ed_routine_idle AND idle.nv_3335_a_idle_request OR general.ed_routine_cip AND nv_3335_a_cip_request OR general.ed_routine_stop AND nv_3335_a_open_request) AND NOT gen_alm_active OR general.ed_routine_manual AND manual_mode.nv_3335_a_manual_request OR general.ed_routine_maint AND maint_mode.nv_3335_a_maint_request) AND NOT stopping_mode.nv_3335_a_stop_request;

// NETWORK 12
nv_3335_a(
    open_feedback := io_mapping.nv_3335_a_open_feedback,
    closed_feedback := io_mapping.nv_3335_a_closed_feedback,
    open_request := nv_3335_a_open_request,
    fault := faults.nv_3335_a_fail_to_close.active OR faults.nv_3335_a_fail_to_open.active); // valve_digital

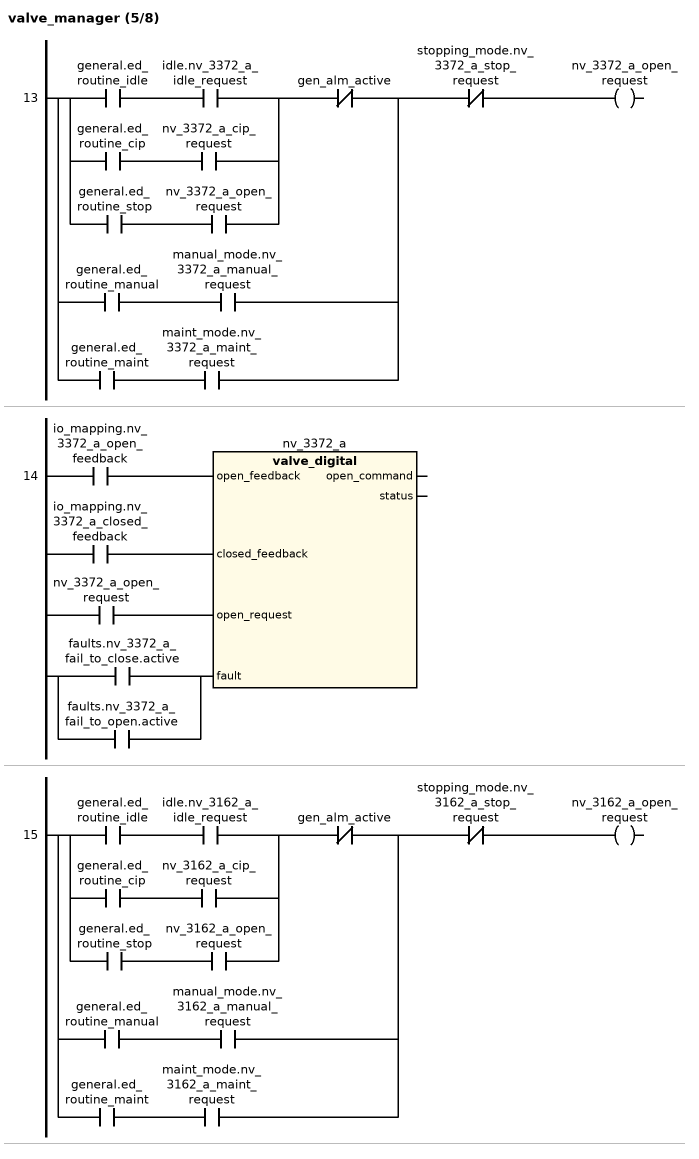
// NETWORK 13
nv_3372_a_open_request := ((general.ed_routine_idle AND idle.nv_3372_a_idle_request OR general.ed_routine_cip AND nv_3372_a_cip_request OR general.ed_routine_stop AND nv_3372_a_open_request) AND NOT gen_alm_active OR general.ed_routine_manual AND manual_mode.nv_3372_a_manual_request OR general.ed_routine_maint AND maint_mode.nv_3372_a_maint_request) AND NOT stopping_mode.nv_3372_a_stop_request;

// NETWORK 14
nv_3372_a(
    open_feedback := io_mapping.nv_3372_a_open_feedback,
    closed_feedback := io_mapping.nv_3372_a_closed_feedback,
    open_request := nv_3372_a_open_request,
    fault := faults.nv_3372_a_fail_to_close.active OR faults.nv_3372_a_fail_to_open.active); // valve_digital

// NETWORK 15
nv_3162_a_open_request := ((general.ed_routine_idle AND idle.nv_3162_a_idle_request OR general.ed_routine_cip AND nv_3162_a_cip_request OR general.ed_routine_stop AND nv_3162_a_open_request) AND NOT gen_alm_active OR general.ed_routine_manual AND manual_mode.nv_3162_a_manual_request OR general.ed_routine_maint AND maint_mode.nv_3162_a_maint_request) AND NOT stopping_mode.nv_3162_a_stop_request;

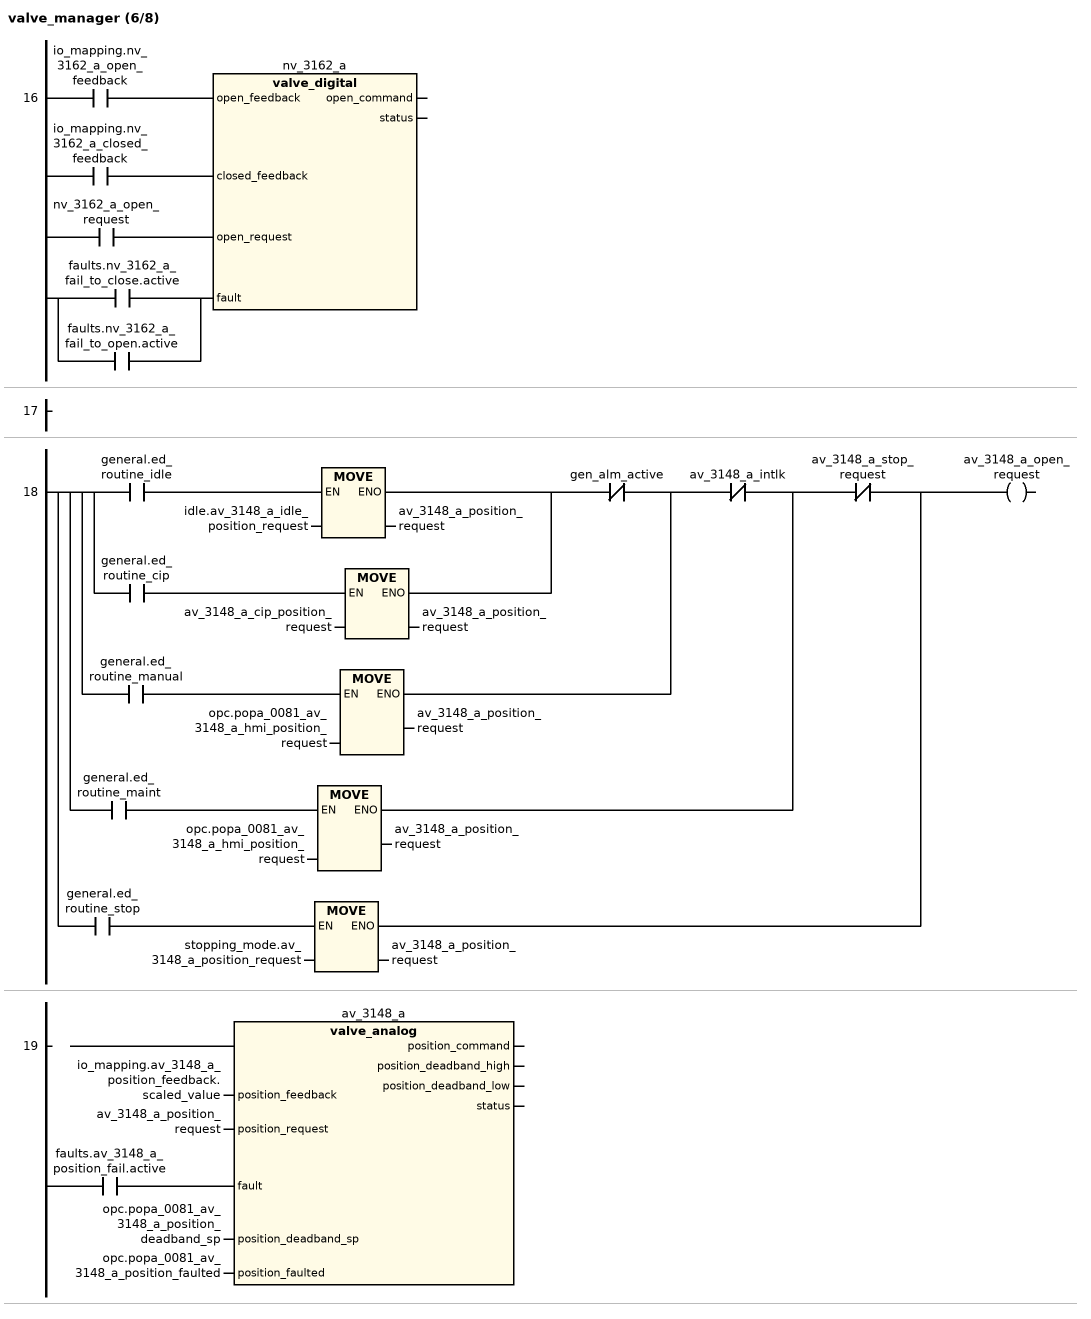
// NETWORK 16
nv_3162_a(
    open_feedback := io_mapping.nv_3162_a_open_feedback,
    closed_feedback := io_mapping.nv_3162_a_closed_feedback,
    open_request := nv_3162_a_open_request,
    fault := faults.nv_3162_a_fail_to_close.active OR faults.nv_3162_a_fail_to_open.active); // valve_digital

// NETWORK 17

// NETWORK 18
_w1 := general.ed_routine_idle;
IF _w1 THEN av_3148_a_position_request := idle.av_3148_a_idle_position_request; END_IF
_w2 := general.ed_routine_cip;
IF _w2 THEN av_3148_a_position_request := av_3148_a_cip_position_request; END_IF
_w3 := general.ed_routine_manual;
IF _w3 THEN av_3148_a_position_request := opc.popa_0081_av_3148_a_hmi_position_request; END_IF
_w4 := general.ed_routine_maint;
IF _w4 THEN av_3148_a_position_request := opc.popa_0081_av_3148_a_hmi_position_request; END_IF
_w5 := general.ed_routine_stop;
IF _w5 THEN av_3148_a_position_request := stopping_mode.av_3148_a_position_request; END_IF
av_3148_a_open_request := (((_w1 OR _w2) AND NOT gen_alm_active OR _w3) AND NOT av_3148_a_intlk OR _w4) AND NOT av_3148_a_stop_request OR _w5;

// NETWORK 19
av_3148_a(
    position_feedback := io_mapping.av_3148_a_position_feedback.scaled_value,
    position_request := av_3148_a_position_request,
    fault := faults.av_3148_a_position_fail.active,
    position_deadband_sp := opc.popa_0081_av_3148_a_position_deadband_sp,
    position_faulted := opc.popa_0081_av_3148_a_position_faulted); // valve_analog

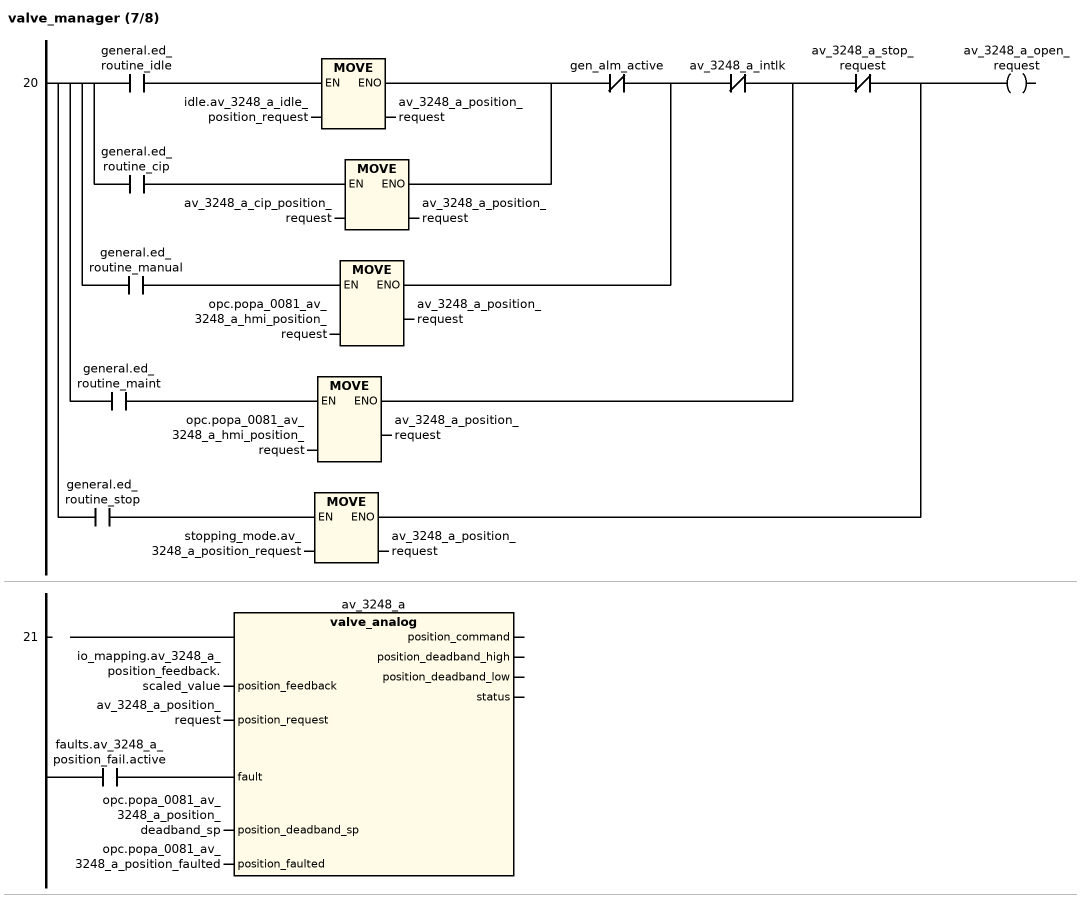
// NETWORK 20
_w6 := general.ed_routine_idle;
IF _w6 THEN av_3248_a_position_request := idle.av_3248_a_idle_position_request; END_IF
_w7 := general.ed_routine_cip;
IF _w7 THEN av_3248_a_position_request := av_3248_a_cip_position_request; END_IF
_w8 := general.ed_routine_manual;
IF _w8 THEN av_3248_a_position_request := opc.popa_0081_av_3248_a_hmi_position_request; END_IF
_w9 := general.ed_routine_maint;
IF _w9 THEN av_3248_a_position_request := opc.popa_0081_av_3248_a_hmi_position_request; END_IF
_w10 := general.ed_routine_stop;
IF _w10 THEN av_3248_a_position_request := stopping_mode.av_3248_a_position_request; END_IF
av_3248_a_open_request := (((_w6 OR _w7) AND NOT gen_alm_active OR _w8) AND NOT av_3248_a_intlk OR _w9) AND NOT av_3248_a_stop_request OR _w10;

// NETWORK 21
av_3248_a(
    position_feedback := io_mapping.av_3248_a_position_feedback.scaled_value,
    position_request := av_3248_a_position_request,
    fault := faults.av_3248_a_position_fail.active,
    position_deadband_sp := opc.popa_0081_av_3248_a_position_deadband_sp,
    position_faulted := opc.popa_0081_av_3248_a_position_faulted); // valve_analog

